	        IF #s_UDT_Status.Specific.ParcelTooLowError
	            OR #iqUDT_EquipmentControl.Command.ResetData
	        THEN
	            "FC_Statistics"(ix_Reset := #iqUDT_EquipmentControl.Command.ResetData,
	                            ix_Activate := #s_UDT_Status.Specific.ParcelTooLowError,
	                            ix_RTrigActivate := #s_R_TRIG_ParcelTooLow.Q,
	                            iqUDT_Statistics := #s_UDT_DimensionsCheckStatistics.TooLowParcels);
	        END_IF;

	    END_REGION

	    REGION 9.5 - Too wide parcels statistics

	        IF #s_UDT_Status.Specific.ParcelTooWideError
	            OR #iqUDT_EquipmentControl.Command.ResetData
	        THEN
	            "FC_Statistics"(ix_Reset := #iqUDT_EquipmentControl.Command.ResetData,
	                            ix_Activate := #s_UDT_Status.Specific.ParcelTooWideError,
	                            ix_RTrigActivate := #s_R_TRIG_ParcelTooWide.Q,
	                            iqUDT_Statistics := #s_UDT_DimensionsCheckStatistics.TooWideParcels);
	        END_IF;

	    END_REGION

	    REGION 9.6 - Too narrow parcels statistics

	        IF #s_UDT_Status.Specific.ParcelTooNarrowError
	            OR #iqUDT_EquipmentControl.Command.ResetData
	        THEN
	            "FC_Statistics"(ix_Reset := #iqUDT_EquipmentControl.Command.ResetData,
	                            ix_Activate := #s_UDT_Status.Specific.ParcelTooNarrowError,
	                            ix_RTrigActivate := #s_R_TRIG_ParcelTooNarrow.Q,
	                            iqUDT_Statistics := #s_UDT_DimensionsCheckStatistics.TooNarrowParcels);
	        END_IF;

	    END_REGION

	    REGION 9.7 - Incorrect parcel orientation statistics

	        IF #s_UDT_Status.Specific.IncorrectParcelOrientationError
	            OR #iqUDT_EquipmentControl.Command.ResetData
	        THEN
	            "FC_Statistics"(ix_Reset := #iqUDT_EquipmentControl.Command.ResetData,
	                            ix_Activate := #s_UDT_Status.Specific.IncorrectParcelOrientationError,
	                            ix_RTrigActivate := #s_R_TRIG_IncorrectShape.Q,
	                            iqUDT_Statistics := #s_UDT_DimensionsCheckStatistics.IncorrectShape);
	        END_IF;

	    END_REGION

	    REGION 9.8 - General error statistics

	        IF #s_UDT_Status.Specific.GeneralError
	            OR #iqUDT_EquipmentControl.Command.ResetData
	        THEN
	            "FC_Statistics"(ix_Reset := #iqUDT_EquipmentControl.Command.ResetData,
	                            ix_Activate := #s_UDT_Status.Specific.GeneralError,
	                            ix_RTrigActivate := #s_R_TRIG_GeneralError.Q,
	                            iqUDT_Statistics := #s_UDT_DimensionsCheckStatistics.GeneralError);
	        END_IF;

	    END_REGION

	END_REGION

	REGION 10 - Status

	    //Status
	    IF #iqUDT_EquipmentControl.Report.EnergySave
	    THEN
	        #s_UDT_Status.Status := "DB_HMIStatusConfiguration".EnergySave;
	    END_IF;

	    IF #iqUDT_EquipmentControl.Report.Running
	    THEN
	        #s_UDT_Status.Status := "DB_HMIStatusConfiguration".Running;
	    END_IF;

	    IF #iqUDT_EquipmentControl.Report.Stopped
	    THEN
	        #s_UDT_Status.Status := "DB_HMIStatusConfiguration".Stopped;
	    END_IF;

	    IF #s_UDT_Status.Specific.ParcelTooLongError
	        OR #s_UDT_Status.Specific.ParcelTooShortError
	        OR #s_UDT_Status.Specific.ParcelTooHighError
	        OR #s_UDT_Status.Specific.ParcelTooLowError
	        OR #s_UDT_Status.Specific.ParcelTooWideError
	        OR #s_UDT_Status.Specific.ParcelTooNarrowError
	        OR #s_UDT_Status.Specific.IncorrectParcelOrientationError
	        OR #s_UDT_Status.Specific.GeneralError

	    THEN
	        #s_UDT_Status.Status := "DB_HMIStatusConfiguration".DimensionError;
	    END_IF;

	(*    IF #iq_UDT_EquipmentControl.Report.SafetyStop
	    THEN
	        #s_UDT_Status.Status := "DB_HMIStatusConfiguration".SafetyStop;
	    END_IF; *)

	END_REGION

	REGION 11 - Update outputs

	    #qUDT_HMIStatus := #s_UDT_Status;
	    #qx_RequestHoldConveyor := (#sx_RequestHold AND NOT #sx_RequestRunReverse) OR #s_UDT_Status.Specific.GeneralError;
	    #qx_RequestRunReverseConveyor := #sx_RequestRunReverse;

	    //Column buzzer
	    #qx_BuzzerColumn := (#sx_ParcelRejecte AND "mx_Clock_1Hz") AND NOT #ix_ReverseRunButton;
	    //Column blue light
	    #qx_LightColumn := (#sx_ParcelRejecte AND "mx_Clock_1Hz") AND NOT #ix_ReverseRunButton;

	    //Button blue light
	    //Steady - Reset and restart line
	    //Blink - Restart not possible, sensor dimensioning check is still covered
	    #qx_LightResetButton := (#sx_ParcelRejecte AND "mx_Clock_1Hz") OR (NOT #sx_ParcelRejecte AND #sx_RequestHold);

	    //Data to HMI
	    //Sensor 1
	    #qUDT_HMIData.ActualSensor1 := #ii_DistanceSensor1;
	    #qUDT_HMIData.OffsetSensor1 := #si_Offset_DistanceSensor1;
	    #qUDT_HMIData.PositionSensor1 := #ii_DistanceSensor1 - #si_Offset_DistanceSensor1;

	    //Sensor 2
	    #qUDT_HMIData.ActualSensor2 := #ii_DistanceSensor2;
	    #qUDT_HMIData.OffsetSensor2 := #si_Offset_DistanceSensor2;
	    #qUDT_HMIData.PositionSensor2 := #ii_DistanceSensor2 - #si_Offset_DistanceSensor2;

	    #qUDT_HMIData.BeltWidth := INT_TO_UINT(#iUDT_DimensionsCheckConfiguration.Position.BeltWidth);


	    IF #s_F_TRIG_WaitForAllScanData.Q THEN
	        IF (#ss_Parcel.Size[0].Width < INT_TO_UINT(#iUDT_DimensionsCheckConfiguration.Position.BeltWidth)) THEN
	            #sui_ProductWidth := #ss_Parcel.Size[0].Width;
	        ELSE
	            #sui_ProductWidth := 0;
	        END_IF;

	        FOR #ti_LoopParcelLength := 0 TO #ci_MeasurementArraySize DO

	            IF (#ss_Parcel.Size[#ti_LoopParcelLength].Width > #sui_ProductWidth) AND (#ss_Parcel.Size[#ti_LoopParcelLength].Width < INT_TO_UINT(#iUDT_DimensionsCheckConfiguration.Position.BeltWidth)) THEN
	                #sui_ProductWidth := #ss_Parcel.Size[#ti_LoopParcelLength].Width;
	            END_IF;

	        END_FOR;

	    END_IF;

	    IF (#sui_ProductWidth > 0)
	        AND (#sui_ProductWidth < #iUDT_DimensionsCheckConfiguration.Position.BeltWidth)
	    THEN

	        #qUDT_HMIData.ProductWidth := #sui_ProductWidth;

	    ELSE

	        #qUDT_HMIData.ProductWidth := 0;

	    END_IF;

	END_REGION

	REGION 12 - Deactivation of functionality

	    #s_UDT_Status.Specific.DisabledGeneralFunctionality := #iUDT_DimensionsCheckCommand.DisableGeneral;
	    #s_UDT_Status.Specific.DisabledTooLongParcel := #iUDT_DimensionsCheckConfiguration.Functionality.TooLongParcelError AND #iUDT_DimensionsCheckCommand.DisableTooLongParcelError;
	    #s_UDT_Status.Specific.DisabledTooShortParcelError := #iUDT_DimensionsCheckConfiguration.Functionality.TooShortParcelError AND #iUDT_DimensionsCheckCommand.DisableTooShortParcelError;
	    #s_UDT_Status.Specific.DisabledTooHighParcelError := #iUDT_DimensionsCheckConfiguration.Functionality.TooHighParcelError AND #iUDT_DimensionsCheckCommand.DisableTooHighParcelError;
	    #s_UDT_Status.Specific.DisabledTooLowParcelError := #iUDT_DimensionsCheckConfiguration.Functionality.TooLowParcelError AND #iUDT_DimensionsCheckCommand.DisableTooLowParcelError;
	    #s_UDT_Status.Specific.DisabledTooWideParcelError := #iUDT_DimensionsCheckConfiguration.Functionality.TooWideParcelError AND #iUDT_DimensionsCheckCommand.DisableTooWideParcelError;
	    #s_UDT_Status.Specific.DisabledTooNarrowParcelError := #iUDT_DimensionsCheckConfiguration.Functionality.TooNarrowParcelError AND #iUDT_DimensionsCheckCommand.DisableTooNarrowParcelError;
	    #s_UDT_Status.Specific.DisabledParcelOrientationError := #iUDT_DimensionsCheckConfiguration.Functionality.ParcelOrientationError AND #iUDT_DimensionsCheckCommand.DisableParcelOrientationError;

	END_REGION
END_FUNCTION_BLOCK

FUNCTION_BLOCK "FB_PECUpdate"
TITLE = FB_PECUpdate
{ S7_Optimized_Access := 'TRUE' }
AUTHOR : MHSE
FAMILY : GeneralSystemFunctions
VERSION : 3.0
// ATTRIBUTES
// AUTO_NUMBER = True
// BLOCK_NUMBER = 221
// END_ATTRIBUTES
//Function block to update parcel data in a tracking array at PEC position.
   VAR_INPUT
      iUDT_PECUpdateConfiguration { ExternalAccessible := 'False'; ExternalVisible := 'False'; ExternalWritable := 'False'} : "UDT_PECUpdateConfiguration";   //   PEC update configuration
      iUDT_ConveyorCommonConfiguration { ExternalAccessible := 'False'; ExternalVisible := 'False'; ExternalWritable := 'False'} : "UDT_ConveyorCommonConfiguration";   //   Conveyor configuration
      ix_PEC { ExternalAccessible := 'False'; ExternalVisible := 'False'; ExternalWritable := 'False'} : Bool;   //   TRUE when the end of section photoeye is not blocked
      ix_TeachingMode { ExternalAccessible := 'False'; ExternalVisible := 'False'; ExternalWritable := 'False'} : Bool;   //   Teaching mode enable
   END_VAR

   VAR_OUTPUT
      qUDT_Status { ExternalAccessible := 'False'; ExternalVisible := 'False'; ExternalWritable := 'False'} : "UDT_PECUpdateStatus";   //   Status structure
      qi_GINwrite { ExternalAccessible := 'False'; ExternalVisible := 'False'; ExternalWritable := 'False'} : Int;   //  Gin found or generated
      qx_PECFiltered { ExternalAccessible := 'False'; ExternalVisible := 'False'; ExternalWritable := 'False'} : Bool;   //   Filtered photoeye signal
   END_VAR

   VAR_IN_OUT
      iqUDT_ConveyorInterface : "UDT_ConveyorInterface";   //   Conveyor interface
      iqUDT_UnknownGINRange : "UDT_UnknownGIN";   //   Unknown GIN
      iqUDT_FifoHeader : "UDT_FifoHeader";   //   FIFO header
      iqUDT_Statistics : "UDT_PECUpdateStatistics";   //   Statistic structure
      iqa_TrackingData : Array[*] of Int;   //   Tracking data
      iqa_FifoData : Array[*] of Int;   //   FIFO data
   END_VAR

   VAR
      sFB_PEC { ExternalAccessible := 'False'; ExternalVisible := 'False'; ExternalWritable := 'False'; S7_SetPoint := 'False'} : "FB_PEC";   //   Photoeye function
      sFB_LengthMeasurement { ExternalAccessible := 'False'; ExternalVisible := 'False'; ExternalWritable := 'False'; S7_SetPoint := 'False'} : "FB_ParcelLength";   //   Length measurement
      sUDT_LostGINFIFOStatus { ExternalAccessible := 'False'; ExternalVisible := 'False'; ExternalWritable := 'False'; S7_SetPoint := 'False'} : "UDT_FifoStatus";   //   Lost GIN FIFO status
      ss_PECDataDeviation { ExternalAccessible := 'False'; ExternalVisible := 'False'; ExternalWritable := 'False'} : Struct   // PEC/Data deviation calculation structure
         Last { ExternalAccessible := 'False'; ExternalVisible := 'False'; ExternalWritable := 'False'} : Int;   //  Last deviation [cm]
         GIN { ExternalAccessible := 'False'; ExternalVisible := 'False'; ExternalWritable := 'False'} : Int;   //  Last GIN deviation
         Sum { ExternalAccessible := 'False'; ExternalVisible := 'False'; ExternalWritable := 'False'} : Int;   //  Deviation sum [cm]
         Nr { ExternalAccessible := 'False'; ExternalVisible := 'False'; ExternalWritable := 'False'} : Int;   //  Deviation number
      END_STRUCT;
      ss_ValidGINRange { ExternalAccessible := 'False'; ExternalVisible := 'False'; ExternalWritable := 'False'} : Struct   //   Valid GIN range
         Start { ExternalAccessible := 'False'; ExternalVisible := 'False'; ExternalWritable := 'False'} : Int;
         End { ExternalAccessible := 'False'; ExternalVisible := 'False'; ExternalWritable := 'False'} : Int;
         GIN { ExternalAccessible := 'False'; ExternalVisible := 'False'; ExternalWritable := 'False'} : Int;
      END_STRUCT;
      ss_AlignedParcelsCounters { ExternalAccessible := 'False'; ExternalVisible := 'False'; ExternalWritable := 'False'} : Struct   //   Aligned parcels counters
         Total { ExternalAccessible := 'False'; ExternalVisible := 'False'; ExternalWritable := 'False'} : Int;   //   Total aligned parcels
         DataNoPEC { ExternalAccessible := 'False'; ExternalVisible := 'False'; ExternalWritable := 'False'} : Int;   //   Parcels aligned in case data detected without photoeye signal
         PECNoData { ExternalAccessible := 'False'; ExternalVisible := 'False'; ExternalWritable := 'False'} : Int;   //   Parcels aligned in case parcel detected without data
      END_STRUCT;
      ss_LostParcelsCounters { ExternalAccessible := 'False'; ExternalVisible := 'False'; ExternalWritable := 'False'} : Struct   //   Lost parcels counters
         Total { ExternalAccessible := 'False'; ExternalVisible := 'False'; ExternalWritable := 'False'} : Int;   //   Total number of lost parcels
         DoubleData { ExternalAccessible := 'False'; ExternalVisible := 'False'; ExternalWritable := 'False'} : Int;   //   Parcels lost due to double data found in a search window
         ParcelNotFound { ExternalAccessible := 'False'; ExternalVisible := 'False'; ExternalWritable := 'False'} : Int;   //   Parcels lost due to no parcel detected after travelling search window distance
      END_STRUCT;
      ss_LostValidParcelsCounters { ExternalAccessible := 'False'; ExternalVisible := 'False'; ExternalWritable := 'False'} : Struct   //   Lost parcels counters
         Total { ExternalAccessible := 'False'; ExternalVisible := 'False'; ExternalWritable := 'False'} : Int;   //   Total number of lost parcels
         DoubleData { ExternalAccessible := 'False'; ExternalVisible := 'False'; ExternalWritable := 'False'} : Int;   //   Parcels lost due to double data found in a search window
         ParcelNotFound { ExternalAccessible := 'False'; ExternalVisible := 'False'; ExternalWritable := 'False'} : Int;   //   Parcels lost due to no parcel detected after travelling search window distance
      END_STRUCT;
      si_UnknownParcelsCounters { ExternalAccessible := 'False'; ExternalVisible := 'False'; ExternalWritable := 'False'} : Struct   //   Unknown parcels counters
         Total { ExternalAccessible := 'False'; ExternalVisible := 'False'; ExternalWritable := 'False'} : Int;   //   Total number of unknown parcels
         LostParcelFound { ExternalAccessible := 'False'; ExternalVisible := 'False'; ExternalWritable := 'False'} : Int;   //   Parcel found with a lost data, unknown GIN created
         DataNotFound { ExternalAccessible := 'False'; ExternalVisible := 'False'; ExternalWritable := 'False'} : Int;   //   Data not found during search window scan
      END_STRUCT;
      sR_TRIG_Parcel {InstructionName := 'R_TRIG'; LibVersion := '1.0'; ExternalAccessible := 'False'; ExternalVisible := 'False'; ExternalWritable := 'False'; S7_SetPoint := 'False'} : R_TRIG;   //   Parcel detected rising edge to count parcels
      sR_TRIG_ParcelFound {InstructionName := 'R_TRIG'; LibVersion := '1.0'; ExternalAccessible := 'False'; ExternalVisible := 'False'; ExternalWritable := 'False'; S7_SetPoint := 'False'} : R_TRIG;   //   Parcel detected rising edge to update the PEC position tracking record
      sR_TRIG_DataFound {InstructionName := 'R_TRIG'; LibVersion := '1.0'; ExternalAccessible := 'False'; ExternalVisible := 'False'; ExternalWritable := 'False'; S7_SetPoint := 'False'} : R_TRIG;   //   Any data found at a PEC position rising edge
      sR_TRIG_PositiveDataFound {InstructionName := 'R_TRIG'; LibVersion := '1.0'; ExternalAccessible := 'False'; ExternalVisible := 'False'; ExternalWritable := 'False'; S7_SetPoint := 'False'} : R_TRIG;   //   Positive data found at a PEC position rising edge
      sR_TRIG_TeachMode {InstructionName := 'R_TRIG'; LibVersion := '1.0'; ExternalAccessible := 'False'; ExternalVisible := 'False'; ExternalWritable := 'False'; S7_SetPoint := 'False'} : R_TRIG;   //   Teaching mode activation rising edge
      sR_TRIG_TooManyLost {InstructionName := 'R_TRIG'; LibVersion := '1.0'; ExternalAccessible := 'False'; ExternalVisible := 'False'; ExternalWritable := 'False'; S7_SetPoint := 'False'} : R_TRIG;   //   Too many lost parcels error statistics trigger
      slr_Performance { ExternalAccessible := 'False'; ExternalVisible := 'False'; ExternalWritable := 'False'} : LReal := 100.0;   //   Update performance [%]
      sdi_TotalNumberOfParcels { ExternalAccessible := 'False'; ExternalVisible := 'False'; ExternalWritable := 'False'} : DInt;   //   Total number of parcels detected
      sdi_TotalNumberOfData { ExternalAccessible := 'False'; ExternalVisible := 'False'; ExternalWritable := 'False'} : DInt;   //   Total number of data detected
      si_PECPosition { ExternalAccessible := 'False'; ExternalVisible := 'False'; ExternalWritable := 'False'} : Int;   //   Photoeye position [cm]
      si_SearchWindow { ExternalAccessible := 'False'; ExternalVisible := 'False'; ExternalWritable := 'False'} : Int;   //   Data search distance from photoeye position [cm]
      si_GINToWrite { ExternalAccessible := 'False'; ExternalVisible := 'False'; ExternalWritable := 'False'} : Int;   //   Found or generated GIN, which will be used to update photoeye position in the tracking array
      si_PositionToUpdate { ExternalAccessible := 'False'; ExternalVisible := 'False'; ExternalWritable := 'False'} : Int;   //   Position in a tracking array to be updated
      si_Direction { ExternalAccessible := 'False'; ExternalVisible := 'False'; ExternalWritable := 'False'} : Int;   //   Direction of the displacement to parametrize loops
      si_Displacement { ExternalAccessible := 'False'; ExternalVisible := 'False'; ExternalWritable := 'False'} : Int;   //   Displacement [cm]
      si_ParcelWaitDistance { ExternalAccessible := 'False'; ExternalVisible := 'False'; ExternalWritable := 'False'} : Int;   //   Parcel delay [cm]
      si_LastUpdatedGIN { ExternalAccessible := 'False'; ExternalVisible := 'False'; ExternalWritable := 'False'} : Int;   //   Last updated GIN to check if next data is a new one
      si_LastCountedData { ExternalAccessible := 'False'; ExternalVisible := 'False'; ExternalWritable := 'False'} : Int;   //   Last counted data
      si_LostParcelsInARow { ExternalAccessible := 'False'; ExternalVisible := 'False'; ExternalWritable := 'False'} : Int;   //   Number of lost parcel in a row
      si_NumberOfTeachedParcels { ExternalAccessible := 'False'; ExternalVisible := 'False'; ExternalWritable := 'False'} : Int;   //   Number of teached parcels
      si_AverageSlip { ExternalAccessible := 'False'; ExternalVisible := 'False'; ExternalWritable := 'False'} : Int;   //   Average parcel slip [cm]
      si_CalculatedLengthCorrection { ExternalAccessible := 'False'; ExternalVisible := 'False'; ExternalWritable := 'False'} : Int;   //   Calculated length correction after teaching
      si_ParcelLengthFilterCounter { ExternalAccessible := 'False'; ExternalVisible := 'False'; ExternalWritable := 'False'} : Int;   //  Parcel length filter counter [cm]
      si_ParcelLengthFilterOldGIN { ExternalAccessible := 'False'; ExternalVisible := 'False'; ExternalWritable := 'False'} : Int;   //  Parcel length filter old GIN
      si_LoopCounter { ExternalAccessible := 'False'; ExternalVisible := 'False'; ExternalWritable := 'False'} : Int;   //   Loop counter
      sx_ParcelDetected { ExternalAccessible := 'False'; ExternalVisible := 'False'; ExternalWritable := 'False'} : Bool;   //   Parcel detected
      sx_ParcelWaitEnable { ExternalAccessible := 'False'; ExternalVisible := 'False'; ExternalWritable := 'False'} : Bool;   //   Missing parcel monitoring
      sx_TeachingMode { ExternalAccessible := 'False'; ExternalVisible := 'False'; ExternalWritable := 'False'} : Bool;   //   Teaching mode
      sx_GenerateGIN { ExternalAccessible := 'False'; ExternalVisible := 'False'; ExternalWritable := 'False'} : Bool;   //   Request to generate GIN
      sx_LostGINFIFOError { ExternalAccessible := 'False'; ExternalVisible := 'False'; ExternalWritable := 'False'} : Bool;   //   Lost GIN FIFO error
      sx_LostGINFIFOWarning { ExternalAccessible := 'False'; ExternalVisible := 'False'; ExternalWritable := 'False'} : Bool;   //   Lost GIN FIFO warning
      sx_InvalidDirection { ExternalAccessible := 'False'; ExternalVisible := 'False'; ExternalWritable := 'False'} : Bool;   //   Invalid direction
      sx_InvalidGINRange { ExternalAccessible := 'False'; ExternalVisible := 'False'; ExternalWritable := 'False'} : Bool;   //   Invalid GIN range
      sx_InvalidDisplacement { ExternalAccessible := 'False'; ExternalVisible := 'False'; ExternalWritable := 'False'} : Bool;   //   Invalid displacement
      sx_InvalidSearchWindow { ExternalAccessible := 'False'; ExternalVisible := 'False'; ExternalWritable := 'False'} : Bool;   //   Invalid search window
      sx_DoubleDataFound { ExternalAccessible := 'False'; ExternalVisible := 'False'; ExternalWritable := 'False'} : Bool;   //   Double data detected
      sx_LengthMeasurementEnable { ExternalAccessible := 'False'; ExternalVisible := 'False'; ExternalWritable := 'False'} : Bool;
   END_VAR

   VAR_TEMP
      tUDT_PECConfiguration : "UDT_PECConfiguration";   //   PEC configuration
      tUDT_PECStatus : "UDT_PECStatus";   //   PEC status
   END_VAR

   VAR CONSTANT
      ci_ZeroGIN : Int;   //   GIN = 0
   END_VAR


BEGIN
	(*
	----------------------------------------------------------------------------------------

	Version history:
	Date        | Version   | Author        | Remark
	----------------------------------------------------------------------------------------
	24/05/2019  | 0.1       | L.Klar        | first release MHSE TIA 15.1
	13/06/2019  | 0.2       | A.Nowak       | Replacement of instruction if for direct write into variable
	21/06/2019  | 0.3       | A.Nowak       | Add gap mesurement function and reorganise block (regions)
	24/07/2019  | 2.0       | L.Klar        | 2.0 MHSE library release TIA 15.1
	23/08/2019  | 2.1       | L.Klar        | "UDT_ConveyorConfiguration" changed to "UDT_ConveyorCommonConfiguration"
	XX/08/2019  | 2.2       | L.Klar        | Update logic changed
	19/09/2019  | 2.3       | P.Majka       | Updating checking PEC and PEC filtered signals
	30/09/2019  | 2.4       | L.Klar        | FB_PEC added, Filtered PEC signal output added
	21/10/2019  | 2.6       | L.Klar        | Configuration UDT chanaged to input, PEC configuration interface input name changed
	23/10/2019  | 2.7       | P.Majka       | Added Region 1, renumerating Regions, changed logic in Region 10.3 and Region 5
	29/10/2019  | 2.8       | L.Klar        | FB_PEC call changed
	14/11/2019  | 2.9       | L.Klar        | Deviations calculation corrected
	14/11/2019  | 3.0       | P.Majka       | 3.0 MHSE library release TIA 15.1
	20/12/2019  | 3.1       | S.Deulkar     | Used configureation error bit to report to conveyor block
	07/01/2020  | 3.2       | L.Klar        | GIN record structure updated, GIN cleared with default one during generation
	                                        | PECUpdate configuration UDT update - search window DINT -> INT,
	                                        | Conveyor common configuration UDT update - length INT -> DINT  conversion added
	29/01/2020  | 3.3       | L.Klar        | Negative GIN handling fixed, configuration bit added to delete negative GIN instead of ignoing it.
	24/02/2020  | 3.4       | L.Klar        | Formating changes, statistics counter added
	10/03/2020  | 3.5       | F.Baten       | Range check unknown GIN region 7
	26/03/2020  | 3.6       | F.Baten       | Added output 'qi_GINwrite'
	25/11/2020  | 3.7       | L.Klar        | Length filter added
	07/12/2020  | 3.8       | L.Klar        | Length filter bug fix
	22/01/2021  | 3.9       | L.Klar        | Total number of parcels and lost parcels counter fixed
	14/08/2021  | 3.10      | S. Deulkar    | Update from EMA
	21/02/2023  | 4.0       | F.Baten       | 4.0 Release TIA 17.5
	*)


	REGION 1 – FIFO header status update

	    "FC_Fifo"(ic_Mode := 'S',
	              qUDT_Status => #sUDT_LostGINFIFOStatus,
	              qx_Error => #sx_LostGINFIFOError,
	              qx_Warning => #sx_LostGINFIFOWarning,
	              iqv_Data := #si_GINToWrite,
	              iqUDT_FifoHeader := #iqUDT_FifoHeader,
	              iqv_DataBuffer := #iqa_FifoData);

	END_REGION

	REGION 2 – Displacement read

	    #si_Displacement := #iqUDT_ConveyorInterface.Displacement;

	END_REGION

	REGION 3 – PEC Position conversion from mm to cm

	    // The conversion is required because the photoeye position is given in mm and the tracking resolution is 1 cm.
	    #si_PECPosition := DINT_TO_INT(#iUDT_PECUpdateConfiguration.Distance / 10);

	END_REGION

	REGION 4 – Teaching mode enable

	    (* Teaching mode is used to calculate conveyor length correction, which allows to align real conveyor length with a tracking array length.
	       Correction is calculated as a difference between photoeye signal and tracking data deviations.
	       Calculated correction has to be manually copied from a FB_PECUpdate instance data block to conveyor configuration.*)

	    // Teaching mode is initialized and activated manually via block input.
	    #sR_TRIG_TeachMode(CLK := #ix_TeachingMode);

	    IF (#sR_TRIG_TeachMode.Q
	        AND NOT #sx_TeachingMode)
	    THEN
	        #ss_PECDataDeviation.Nr := 0;
	        #ss_PECDataDeviation.Sum := 0;
	        #si_NumberOfTeachedParcels := 0;
	        #sx_TeachingMode := TRUE;
	    END_IF;

	END_REGION

	REGION 5 – Photoeye

	    (*FB_PEC block call to filter photoeye signal and calculate jam status.*)

	    // Copy PEC configuration.
	    #tUDT_PECConfiguration.Distance := #iUDT_PECUpdateConfiguration.Distance;
	    #tUDT_PECConfiguration.JamDisplacementLimit := #iUDT_PECUpdateConfiguration.JamDisplacementLimit;
	    #tUDT_PECConfiguration.TimeOnDelay := #iUDT_PECUpdateConfiguration.TimeOnDelay;
	    #tUDT_PECConfiguration.TimeOffDelay := #iUDT_PECUpdateConfiguration.TimeOffDelay;
	    #tUDT_PECConfiguration.ResetWithPECBlocked := #iUDT_PECUpdateConfiguration.ResetWithPECBlocked;

	    //Call FB_PEC.
	    #sFB_PEC(ix_PEC := #ix_PEC,
	             iUDT_PECConfiguration := #tUDT_PECConfiguration,
	             qUDT_HMIStatus => #tUDT_PECStatus,
	             iqUDT_ConveyorInterface := #iqUDT_ConveyorInterface,
	             iqUDT_PECStatistics := #iqUDT_Statistics.PEC);

	    // Parcel length filter
	    IF NOT #ix_PEC
	        AND #iUDT_PECUpdateConfiguration.ParcelLengthFilter
	        AND #iqa_TrackingData[#si_PECPosition - 1] > 0
	        AND #iqa_TrackingData[#si_PECPosition - 1] <> #si_ParcelLengthFilterOldGIN THEN

	        IF "DB_GIN".GIN[#iqa_TrackingData[#si_PECPosition - 1]].General.Length > 0 THEN
	            #si_ParcelLengthFilterCounter := "DB_GIN".GIN[#iqa_TrackingData[#si_PECPosition - 1]].General.Length;
	        END_IF;

	        #si_ParcelLengthFilterOldGIN := #iqa_TrackingData[#si_PECPosition - 1];

	    END_IF;

	    IF #si_ParcelLengthFilterCounter > 0 THEN

	        #qUDT_Status.PEC := FALSE;
	        #qx_PECFiltered := FALSE;
	        #si_ParcelLengthFilterCounter -= #iqUDT_ConveyorInterface.Displacement;

	    ELSE

	        #qUDT_Status.PEC := #sFB_PEC.qx_PECFiltered;
	        #qx_PECFiltered := #sFB_PEC.qx_PECFiltered;

	    END_IF;

	    #qUDT_Status.Jam := #tUDT_PECStatus.Jam;

	    // Parcel detected variable to simplify further photoeye position tracking record update.
	    #sx_ParcelDetected := NOT #qUDT_Status.PEC;

	END_REGION

	REGION 6 – Error reset

	    // Reset errors when reset signal is given.
	    IF (#iqUDT_ConveyorInterface.InternalErrorReset)
	    THEN
	        #si_LostParcelsInARow := 0;
	        #qUDT_Status.TooManyLost := FALSE;
	        #sx_InvalidDisplacement := FALSE;
	    END_IF;

	END_REGION

	REGION 7 – GIN generator initialization

	    // Valid GIN range configuration is moved to a structure.
	    #ss_ValidGINRange.Start := #iUDT_PECUpdateConfiguration.GINRangeStart;
	    #ss_ValidGINRange.End := #iUDT_PECUpdateConfiguration.GINRangeEnd;

	    // Check if the unknown GIN is within range
	    IF #iqUDT_UnknownGINRange.GIN < #iqUDT_UnknownGINRange.Start
	        OR #iqUDT_UnknownGINRange.GIN > #iqUDT_UnknownGINRange.End
	    THEN
	        #iqUDT_UnknownGINRange.GIN := #iqUDT_UnknownGINRange.Start;
	    END_IF;

	    // Whenever valid GIN range is changed and the generated GIN doesn't fit, it's initialized.
	    IF (#ss_ValidGINRange.GIN < #ss_ValidGINRange.Start
	        OR #ss_ValidGINRange.GIN > #ss_ValidGINRange.End)
	    THEN
	        #ss_ValidGINRange.GIN := #ss_ValidGINRange.Start;
	    END_IF;

	    // Valid GIN range is set locally in PEC update configuration structure and it can't overlap with a global unknown GIN range.
	    #sx_InvalidGINRange := #iUDT_PECUpdateConfiguration.GenerationPoint
	    AND (#ss_ValidGINRange.End <= #ss_ValidGINRange.Start
	    OR #ss_ValidGINRange.Start <= #iqUDT_UnknownGINRange.End
	    OR #iqUDT_UnknownGINRange.End <= #iqUDT_UnknownGINRange.Start)
	    AND #ss_ValidGINRange.Start < 1000;   // Until 1000 it is UFO range

	END_REGION

	REGION 8 – Search window and displacement validation

	    (*Both parameters have to be checked to prevent tracking array exceeding.*)

	    // Search window cannot be lower than zero and greater than distance between PEC position and conveyor edge.
	    #sx_InvalidSearchWindow := #iUDT_PECUpdateConfiguration.SearchWindowFwd < 0
	    OR #iUDT_PECUpdateConfiguration.SearchWindowFwd >= #iUDT_ConveyorCommonConfiguration.Length + #iUDT_ConveyorCommonConfiguration.LengthCorrection - #si_PECPosition
	    OR #iUDT_PECUpdateConfiguration.SearchWindowRvs < 0
	    OR #iUDT_PECUpdateConfiguration.SearchWindowRvs >= #si_PECPosition;

	    // Displacement cannot be greater than the photoeye position.
	    IF (ABS(#si_Displacement) > #si_PECPosition)
	    THEN
	        #sx_InvalidDisplacement := TRUE;
	    END_IF;

	END_REGION

	REGION 9 – Total number of parcels counter

	    (*Parcels are counted basing on parcel detection rising edge trigger. Counting is blocked
	      during PLC first scan, when photoeye signal becomes 0.*)

	    #sR_TRIG_Parcel(CLK := #sx_ParcelDetected);

	    IF (#sR_TRIG_Parcel.Q
	        AND NOT "DB_Memory".FirstScan)
	    THEN
	        // Total number of parcels.
	        #sdi_TotalNumberOfParcels += 1;

	        // Every detected parcel resets lost parcels in a row counter.
	        #si_LostParcelsInARow := 0;

	        // Number of teached parcels is incremented if teaching mode is activated.
	        IF (#sx_TeachingMode)
	        THEN
	            #si_NumberOfTeachedParcels += 1;
	        END_IF;
	    END_IF;

	END_REGION

	REGION 10 – PEC Update
	    (* Photoeye position record is updated after every tracking register shift, basing on
	       actual situation - photoeye signal and data availability. In case of displacement
	       graeter than one, the loop will be executed the proper number of times. The update loop
	       can be executed if there is no configuration errors and the displacement was given.*)

	    WHILE #si_Displacement <> 0
	        AND NOT #sx_InvalidGINRange
	        AND NOT #sx_InvalidDisplacement
	        AND NOT #sx_InvalidSearchWindow
	    DO

	        REGION 10.1 – Direction

	            (*Depending on displacement sign, the direction of movement is determinated. This allows to choose
	            ` correct search window and parametrize all search loops to count up or down.*)

	            IF (#si_Displacement < 0)
	            THEN
	                #si_Direction := -1;
	                #si_SearchWindow := #iUDT_PECUpdateConfiguration.SearchWindowRvs;
	            ELSIF (#si_Displacement > 0)
	            THEN
	                #si_Direction := 1;
	                #si_SearchWindow := #iUDT_PECUpdateConfiguration.SearchWindowFwd;
	            END_IF;

	        END_REGION

	        REGION 10.2 – Position to update

	            // Position pointer used to specify the tracking array record to be updated.
	            #si_PositionToUpdate := #si_PECPosition - #si_Displacement + #si_Direction;

	        END_REGION


	        REGION 10.3 – Total number of data counter

	            (*Total number of data is incremented every time when new GIN is detected.*)

	            IF (#iqa_TrackingData[#si_PositionToUpdate + 1] > 0
	                AND #iqa_TrackingData[#si_PositionToUpdate + 1] <> #si_LastCountedData)
	            THEN
	                #sdi_TotalNumberOfData += 1;
	                #si_LastCountedData := #iqa_TrackingData[#si_PositionToUpdate + 1];
	            END_IF;

	        END_REGION

	        REGION 10.4 – GIN detection

	            (* Data found and parcel found triggers are used to determine the update case,
	               whether the data occurred first or a parcel.*)

	            // Trigger on any data found at a PEC position to detect the front of the parcel data.
	            #sR_TRIG_DataFound(CLK := #iqa_TrackingData[#si_PositionToUpdate] <> 0);

	            // Trigger on positive data found at a PEC position to detect the front of the parcel data.
	            #sR_TRIG_PositiveDataFound(CLK := #iqa_TrackingData[#si_PositionToUpdate] > 0);

	            // Trigger to detect front of the parcel.
	            #sR_TRIG_ParcelFound(CLK := #sx_ParcelDetected);

	(*
	Data detected without PEC signal

	                         Search window
	                          <--------|
	Data                              PEC
	|----------------------------------|------------------------------------------|
	|                           XXXXXXXX                                          |
	|----------------------------------|------------------------------------------|
	                                   |
	Conveyor                           |
	|----------------------------------|------------------------------------------|
	|                      YYYYYYYY    |                                          |
	|                      YYYYYYYY    |                                          |
	|                      YYYYYYYY    |                                          |
	|----------------------------------|------------------------------------------|
	*)
	(* Data detected without PEC signal.*)
	            IF (#sR_TRIG_PositiveDataFound.Q
	                AND NOT #sx_ParcelDetected)
	            THEN
	                #si_GINToWrite := 0;
	                // Double data detection loop.
	                FOR #si_LoopCounter := #si_PositionToUpdate TO
	                    #si_PECPosition + (#si_SearchWindow * #si_Direction) BY #si_Direction DO
	                    // Data found in a search window.
	                    IF (#iqa_TrackingData[#si_LoopCounter] > 0)
	                    THEN
	                        // First GIN found.
	                        IF (#si_GINToWrite = 0)
	                        THEN
	                            // Get the GIN if it's different than last updated GIN.
	                            IF #iqa_TrackingData[#si_LoopCounter] <> #si_LastUpdatedGIN THEN
	                                #si_GINToWrite := #iqa_TrackingData[#si_LoopCounter];
	                            END_IF;
	                            // If the first GIN was found, the scan loop conitues to check if there is no other data.
	                        ELSE
	                            // Next found data is different than the first one. Double data detected.
	                            IF (#iqa_TrackingData[#si_LoopCounter] <> #si_GINToWrite)
	                            THEN
	                                #sx_DoubleDataFound := TRUE;
	                                // First found GIN is marked as a lost one and the GIN is stored in a FIFO register.
	                                IF ("DB_GIN".GIN[#si_GINToWrite].General.Lost = FALSE)
	                                THEN
	                                    "DB_GIN".GIN[#si_GINToWrite].General.Lost := TRUE;

	                                    "FC_Fifo"(ic_Mode := 'W',
	                                              qUDT_Status => #sUDT_LostGINFIFOStatus,
	                                              qx_Error => #sx_LostGINFIFOError,
	                                              qx_Warning => #sx_LostGINFIFOWarning,
	                                              iqv_Data := #si_GINToWrite,
	                                              iqUDT_FifoHeader := #iqUDT_FifoHeader,
	                                              iqv_DataBuffer := #iqa_FifoData);

	                                    // Update statistics
	                                    #ss_LostParcelsCounters.Total += 1;
	                                    #ss_LostParcelsCounters.DoubleData += 1;


	                                    ////////////////////

	                                    IF #si_GINToWrite >= 1000 THEN
	                                        #ss_LostValidParcelsCounters.Total += 1;
	                                        #ss_LostValidParcelsCounters.DoubleData += 1;
	                                    END_IF;

	                                    ////////////////
	                                END_IF;

	                                // Second found GIN is marked as a lost one and the GIN is stored in a FIFO register.
	                                IF ("DB_GIN".GIN[#iqa_TrackingData[#si_LoopCounter]].General.Lost = FALSE)
	                                THEN
	                                    "DB_GIN".GIN[#iqa_TrackingData[#si_LoopCounter]].General.Lost := TRUE;

	                                    "FC_Fifo"(ic_Mode := 'W',
	                                              qUDT_Status => #sUDT_LostGINFIFOStatus,
	                                              qx_Error => #sx_LostGINFIFOError,
	                                              qx_Warning => #sx_LostGINFIFOWarning,
	                                              iqv_Data := #iqa_TrackingData[#si_LoopCounter],
	                                              iqUDT_FifoHeader := #iqUDT_FifoHeader,
	                                              iqv_DataBuffer := #iqa_FifoData);

	                                    // Update statistics
	                                    #ss_LostParcelsCounters.Total += 1;
	                                    #ss_LostParcelsCounters.DoubleData += 1;

	                                    ////////////////////

	                                    IF #iqa_TrackingData[#si_LoopCounter] >= 1000 THEN
	                                        #ss_LostValidParcelsCounters.Total += 1;
	                                        #ss_LostValidParcelsCounters.DoubleData += 1;
	                                    END_IF;

	                                    ////////////////
	                                    //
	                                END_IF;
	                                // Stop search window scan in case of double data detection
	                                EXIT;
	                            END_IF;
	                        END_IF;
	                    END_IF;
	                END_FOR;

	                // Becasue the data was found as a first one, GIN is stored and the logic to wait for a parcel is enebaled.
	                // If the double data was found there is no need to wait for a parcel. Data has been marked as a lost one.
	                IF NOT #sx_DoubleDataFound
	                THEN
	                    #sx_ParcelWaitEnable := TRUE;
	                END_IF;

	                #sx_DoubleDataFound := FALSE;
	(*
	Data and PEC signal detected at the same time - perfect match

	                         Search window
	                          <--------|
	Data                              PEC
	|----------------------------------|------------------------------------------|
	|                           XXXXXXXX                                          |
	|----------------------------------|------------------------------------------|
	                                   |
	Conveyor                           |
	|----------------------------------|------------------------------------------|
	|                           XXXXXXXX                                          |
	|                           XXXXXXXX                                          |
	|                           XXXXXXXX                                          |
	|----------------------------------|------------------------------------------|

	or PEC signal found without data or with old ones

	                         Search window
	                          <--------|
	Data                              PEC
	|----------------------------------|------------------------------------------|
	|                    XXXXXXXX      |                                          |
	|----------------------------------|------------------------------------------|
	                                   |
	Conveyor                           |
	|----------------------------------|------------------------------------------|
	|                           XXXXXXXX                                          |
	|                           XXXXXXXX                                          |
	|                           XXXXXXXX                                          |
	|----------------------------------|------------------------------------------|
	*)
	(*Data and PEC signal detected at the same time (perfect match) or PEC signal found without data or with old ones.*)
	            ELSIF (#sR_TRIG_ParcelFound.Q
	                AND (#sR_TRIG_PositiveDataFound.Q
	                OR (#iqa_TrackingData[#si_PositionToUpdate] = 0
	                OR #iqa_TrackingData[#si_PositionToUpdate] = #si_LastUpdatedGIN)
	                AND NOT #sx_ParcelWaitEnable))
	            THEN
	                // If the PEC is set as a GIN generation point, skip data detection loop and go to GIN generator.
	                IF (#iUDT_PECUpdateConfiguration.GenerationPoint)
	                THEN
	                    #sx_GenerateGIN := TRUE;
	                    // If the the PEC isn't a generation point, data search loop is enabled.
	                ELSE
	                    #si_GINToWrite := 0;

	                    // Double data detection loop.
	                    FOR #si_LoopCounter := #si_PositionToUpdate TO
	                        #si_PECPosition + (#si_SearchWindow * #si_Direction) BY #si_Direction DO

	                        // Data found in a search window.
	                        IF (#iqa_TrackingData[#si_LoopCounter] > 0)
	                        THEN
	                            // First GIN found.
	                            IF (#si_GINToWrite = 0)
	                            THEN
	                                // Get the GIN if it's different than last updated GIN.
	                                IF #iqa_TrackingData[#si_LoopCounter] <> #si_LastUpdatedGIN THEN
	                                    #si_GINToWrite := #iqa_TrackingData[#si_LoopCounter];

	                                    // PEC/Data deviation acquisition
	                                    #ss_PECDataDeviation.Last := DINT_TO_INT(#si_PECPosition - #si_LoopCounter);
	                                    #ss_PECDataDeviation.GIN := #si_GINToWrite;
	                                    #ss_PECDataDeviation.Sum -= ABS(#ss_PECDataDeviation.Last);
	                                    #ss_PECDataDeviation.Nr += 1;

	                                    // Parcel aligned statistics
	                                    IF (ABS(#ss_PECDataDeviation.Last) > ABS(#si_Displacement - 1))
	                                    THEN
	                                        #ss_AlignedParcelsCounters.Total += 1;
	                                        #ss_AlignedParcelsCounters.PECNoData += 1;
	                                    END_IF;
	                                END_IF;
	                                // If the first GIN was found, the scan loop conitues to check if there is no other data.
	                            ELSE
	                                // Next found data is different than the first one. Double data detected.
	                                IF (#iqa_TrackingData[#si_LoopCounter] <> #si_GINToWrite)
	                                THEN
	                                    // First found GIN is marked as a lost one and the GIN is stored in a FIFO register.
	                                    IF ("DB_GIN".GIN[#si_GINToWrite].General.Lost = FALSE)
	                                    THEN
	                                        "DB_GIN".GIN[#si_GINToWrite].General.Lost := TRUE;
	                                        "FC_Fifo"(ic_Mode := 'W',
	                                                  qUDT_Status => #sUDT_LostGINFIFOStatus,
	                                                  qx_Error => #sx_LostGINFIFOError,
	                                                  qx_Warning => #sx_LostGINFIFOWarning,
	                                                  iqv_Data := #si_GINToWrite,
	                                                  iqUDT_FifoHeader := #iqUDT_FifoHeader,
	                                                  iqv_DataBuffer := #iqa_FifoData);

	                                        // Update statistics
	                                        #ss_LostParcelsCounters.Total += 1;
	                                        #ss_LostParcelsCounters.DoubleData += 1;

	                                        ////////////////////

	                                        IF #si_GINToWrite >= 1000 THEN
	                                            #ss_LostValidParcelsCounters.Total += 1;
	                                            #ss_LostValidParcelsCounters.DoubleData += 1;
	                                        END_IF;

	                                        ////////////////
	                                        //
	                                    END_IF;

	                                    // Second found GIN is marked as a lost one and the GIN is stored in a FIFO register.
	                                    IF ("DB_GIN".GIN[#iqa_TrackingData[#si_LoopCounter]].General.Lost = FALSE)
	                                    THEN
	                                        "DB_GIN".GIN[#iqa_TrackingData[#si_LoopCounter]].General.Lost := TRUE;
	                                        "FC_Fifo"(ic_Mode := 'W',
	                                                  qUDT_Status => #sUDT_LostGINFIFOStatus,
	                                                  qx_Error => #sx_LostGINFIFOError,
	                                                  qx_Warning => #sx_LostGINFIFOWarning,
	                                                  iqv_Data := #iqa_TrackingData[#si_LoopCounter],
	                                                  iqUDT_FifoHeader := #iqUDT_FifoHeader,
	                                                  iqv_DataBuffer := #iqa_FifoData);

	                                        // Update statistics
	                                        #ss_LostParcelsCounters.Total += 1;
	                                        #ss_LostParcelsCounters.DoubleData += 1;

	                                        ////////////////////

	                                        IF #iqa_TrackingData[#si_LoopCounter] >= 1000 THEN
	                                            #ss_LostValidParcelsCounters.Total += 1;
	                                            #ss_LostValidParcelsCounters.DoubleData += 1;
	                                        END_IF;

	                                        ////////////////
	                                        //
	                                    END_IF;
	                                    // Stop search window scan in case of double data detection
	                                    EXIT;
	                                END_IF;
	                            END_IF;
	                        END_IF;
	                    END_FOR;

	                    // GIN not found in a search window
	                    IF (#si_GINToWrite = 0)
	                    THEN
	                        #sx_GenerateGIN := TRUE;
	                        #si_UnknownParcelsCounters.DataNotFound += 1;
	                    END_IF;

	                    // Found GIN is a lost one - generate unknown GIN
	                    // Found GIN isn't lost or it's negative - don't do anything
	                    IF (#si_GINToWrite > 0)
	                    THEN
	                        IF ("DB_GIN".GIN[#si_GINToWrite].General.Lost)
	                        THEN
	                            #sx_GenerateGIN := TRUE;
	                            #si_UnknownParcelsCounters.LostParcelFound += 1;
	                        END_IF;
	                    END_IF;
	                END_IF;

	                (*Second parcel has been found during data update. Situation can occur when search window is too short
	                  and the data is shifted. In that case found GIN will be marked as a lost one and new unknown GIN will be
	                  generated. Negative GIN will be ignored.*)
	            ELSIF (#sR_TRIG_ParcelFound.Q
	                AND (#iqa_TrackingData[#si_PositionToUpdate] <> 0
	                AND #iqa_TrackingData[#si_PositionToUpdate] <> #si_LastUpdatedGIN)
	                AND NOT #sx_ParcelWaitEnable)
	            THEN
	                IF (#iqa_TrackingData[#si_PositionToUpdate] > 0)
	                THEN
	                    IF ("DB_GIN".GIN[#iqa_TrackingData[#si_PositionToUpdate]].General.Lost = FALSE)
	                    THEN
	                        "DB_GIN".GIN[#iqa_TrackingData[#si_PositionToUpdate]].General.Lost := TRUE;
	                        "FC_Fifo"(ic_Mode := 'W',
	                                  qUDT_Status => #sUDT_LostGINFIFOStatus,
	                                  qx_Error => #sx_LostGINFIFOError,
	                                  qx_Warning => #sx_LostGINFIFOWarning,
	                                  iqv_Data := #iqa_TrackingData[#si_PositionToUpdate],
	                                  iqUDT_FifoHeader := #iqUDT_FifoHeader,
	                                  iqv_DataBuffer := #iqa_FifoData);

	                        // Update statistics
	                        #ss_LostParcelsCounters.Total += 1;
	                        #ss_LostParcelsCounters.DoubleData += 1;

	                        ////////////////////

	                        IF #iqa_TrackingData[#si_PositionToUpdate] >= 1000 THEN
	                            #ss_LostValidParcelsCounters.Total += 1;
	                            #ss_LostValidParcelsCounters.DoubleData += 1;
	                        END_IF;

	                        ////////////////
	                        //
	                    END_IF;
	                END_IF;

	                // Generate GIN
	                #sx_GenerateGIN := TRUE;
	                #si_UnknownParcelsCounters.LostParcelFound += 1;

	                (*Second data has been found during data update. Situation can occur when search window is too short
	                  and the data is shifted. In that case found GIN will be marked as a lost one.*)
	            ELSIF (#sR_TRIG_PositiveDataFound.Q
	                AND #sx_ParcelDetected
	                AND #iqa_TrackingData[#si_PositionToUpdate] <> #si_GINToWrite)
	            THEN
	                // Mark GIN as a lost one
	                IF ("DB_GIN".GIN[#iqa_TrackingData[#si_PositionToUpdate]].General.Lost = FALSE)
	                THEN
	                    "DB_GIN".GIN[#iqa_TrackingData[#si_PositionToUpdate]].General.Lost := TRUE;
	                    "FC_Fifo"(ic_Mode := 'W',
	                              qUDT_Status => #sUDT_LostGINFIFOStatus,
	                              qx_Error => #sx_LostGINFIFOError,
	                              qx_Warning => #sx_LostGINFIFOWarning,
	                              iqv_Data := #iqa_TrackingData[#si_PositionToUpdate],
	                              iqUDT_FifoHeader := #iqUDT_FifoHeader,
	                              iqv_DataBuffer := #iqa_FifoData);

	                    // Update statistics
	                    #ss_LostParcelsCounters.Total += 1;
	                    #ss_LostParcelsCounters.DoubleData += 1;

	                    ////////////////////

	                    IF #iqa_TrackingData[#si_PositionToUpdate] >= 1000 THEN
	                        #ss_LostValidParcelsCounters.Total += 1;
	                        #ss_LostValidParcelsCounters.DoubleData += 1;
	                    END_IF;

	                    ////////////////
	                END_IF;
	            END_IF;

	        END_REGION

	        REGION 10.5 – GIN generator

	            (*Used to generate new GIN. If the PEC position is a generation point, the number is taken from an internal GIN range.
	              If it's not, then GIN is taken from a global unknown GIN range.*)

	            IF (#sx_GenerateGIN)
	            THEN
	                // Generation point.
	                IF (#iUDT_PECUpdateConfiguration.GenerationPoint)
	                THEN
	                    // Generate GIN from a valid GIN range.
	                    IF (#ss_ValidGINRange.GIN <= #ss_ValidGINRange.End)
	                    THEN
	                        #si_GINToWrite := #ss_ValidGINRange.GIN;
	                        #ss_ValidGINRange.GIN += 1;
	                    ELSE
	                        #si_GINToWrite := #ss_ValidGINRange.Start;
	                        #ss_ValidGINRange.GIN := #ss_ValidGINRange.Start + 1;
	                    END_IF;
	                    // Unknown GIN generator.
	                ELSE
	                    // Generate GIN from a unknown GIN range.
	                    IF (#iqUDT_UnknownGINRange.GIN <= #iqUDT_UnknownGINRange.End)
	                    THEN
	                        #si_GINToWrite := #iqUDT_UnknownGINRange.GIN;
	                        #iqUDT_UnknownGINRange.GIN += 1;
	                    ELSE
	                        #si_GINToWrite := #iqUDT_UnknownGINRange.Start;
	                        #iqUDT_UnknownGINRange.GIN := #iqUDT_UnknownGINRange.Start + 1;
	                    END_IF;

	                    // Unknwn parcels statistics.
	                    #si_UnknownParcelsCounters.Total += 1;
	                END_IF;

	                // Reset generte GIN command.
	                #sx_GenerateGIN := FALSE;

	                // GIN record is cleared with configured default GIN record while it's generated.
	                "DB_GIN".GIN[#si_GINToWrite] := "DB_GINDefault".GIN[#iUDT_PECUpdateConfiguration.DefaultGIN];
	            END_IF;

	            #qi_GINwrite := #si_GINToWrite;

	        END_REGION


	        REGION 10.6 – PEC position data update

	            (*While parcel is detected, calculated GIN is written into the PEC position record.
	              If not, then the record is cleared with 0. Negative GIN is ignored or deleted, depending on configuration.*)

	            IF (#sx_ParcelDetected)
	            THEN

	                "FC_WriteGIN"(ii_GIN := #si_GINToWrite,
	                              ii_PositionToWrite := #si_PositionToUpdate,
	                              ii_NumberOfPositions := 1,
	                              ix_Direction := TRUE,
	                              iqa_TrackingData := #iqa_TrackingData);

	            ELSE
	                IF (#iqa_TrackingData[#si_PositionToUpdate] > 0
	                    OR #iUDT_PECUpdateConfiguration.NegativeGINDelete)
	                THEN

	                    "FC_WriteGIN"(ii_GIN := #ci_ZeroGIN,
	                                  ii_PositionToWrite := #si_PositionToUpdate,
	                                  ii_NumberOfPositions := 1,
	                                  ix_Direction := TRUE,
	                                  iqa_TrackingData := #iqa_TrackingData);

	                END_IF;
	            END_IF;

	        END_REGION

	        REGION 10.7 – Parcel waiting logic

	            (*Parcel waiting logic is used to wait for the photoeye signal for a search window distance.*)
	            IF (#sx_ParcelWaitEnable)
	            THEN
	                // Counting parcel wait distance depending on conveyor running direction if not detected.
	                IF (NOT #sx_ParcelDetected)
	                THEN
	                    IF (#si_Direction = 1)
	                    THEN
	                        #si_ParcelWaitDistance += 1;
	                    ELSE
	                        #si_ParcelWaitDistance -= 1;
	                    END_IF;

	                    // Parcel detected - stop waiting, use found GIN to update.
	                ELSE
	                    // PEC/Data deviation acquisition
	                    #ss_PECDataDeviation.Last := #si_ParcelWaitDistance;
	                    #ss_PECDataDeviation.GIN := #si_GINToWrite;
	                    #ss_PECDataDeviation.Sum += ABS(#ss_PECDataDeviation.Last);
	                    #ss_PECDataDeviation.Nr += 1;


	                    // Parcel aligned statistics
	                    IF (#ss_PECDataDeviation.Last > ABS(#si_Displacement - 1))
	                    THEN
	                        #ss_AlignedParcelsCounters.Total += 1;
	                        #ss_AlignedParcelsCounters.DataNoPEC += 1;
	                    END_IF;

	                    // Parcel waiting logic reset.
	                    #sx_ParcelWaitEnable := FALSE;
	                    #si_ParcelWaitDistance := 0;
	                END_IF;
	            END_IF;

	            // Parcel not found in a search window - stop waiting, mark found GIN as a lost one.
	            IF (ABS(#si_ParcelWaitDistance) = #si_SearchWindow)
	                AND (#si_GINToWrite > 0)
	            THEN
	                // Parcel lost
	                IF "DB_GIN".GIN[#si_GINToWrite].General.Lost = FALSE THEN
	                    "DB_GIN".GIN[#si_GINToWrite].General.Lost := TRUE;
	                    "FC_Fifo"(ic_Mode := 'W',
	                              qUDT_Status => #sUDT_LostGINFIFOStatus,
	                              qx_Error => #sx_LostGINFIFOError,
	                              qx_Warning => #sx_LostGINFIFOWarning,
	                              iqv_Data := #si_GINToWrite,
	                              iqUDT_FifoHeader := #iqUDT_FifoHeader,
	                              iqv_DataBuffer := #iqa_FifoData);

	                    // Parcel waiting logic reset.
	                    #si_ParcelWaitDistance := 0;
	                    #sx_ParcelWaitEnable := FALSE;

	                    // Lost parcels ina  row counter.
	                    #si_LostParcelsInARow += 1;

	                    // Update statistics.
	                    #ss_LostParcelsCounters.Total += 1;
	                    #ss_LostParcelsCounters.ParcelNotFound += 1;

	                    ////////////////////

	                    IF #si_GINToWrite >= 1000 THEN
	                        #ss_LostValidParcelsCounters.Total += 1;
	                        #ss_LostValidParcelsCounters.ParcelNotFound += 1;
	                    END_IF;

	                    ////////////////
	                    //
	                END_IF;

	            END_IF;

	            // Reset monitoring in case of going backwards.
	            IF (#si_ParcelWaitDistance = 0
	                AND NOT #sx_ParcelDetected
	                AND #sx_InvalidDirection)
	            THEN
	                #sx_ParcelWaitEnable := FALSE;
	            END_IF;

	            #sx_InvalidDirection := ((#si_Direction = 1
	            AND #si_ParcelWaitDistance < 0)
	            OR (#si_Direction = -1
	            AND #si_ParcelWaitDistance > 0));

	        END_REGION

	        REGION 10.8 – Last updated GIN

	            (*Last updated GIN to avoid processing the same data.*)
	            IF (#sR_TRIG_DataFound.Q)
	            THEN
	                #si_LastUpdatedGIN := #iqa_TrackingData[#si_PositionToUpdate];
	            END_IF;

	        END_REGION

	        REGION 10.8 – Update displacement

	            #si_Displacement := #si_Displacement - #si_Direction;

	        END_REGION

	    END_WHILE;

	END_REGION

	REGION 11 – Length measurement



	    (*Length and gap measurements can be enabled via PEC update configuration*)
	    #sFB_LengthMeasurement(ii_PECPosition := #si_PECPosition,
	                           ii_Displacement := #iqUDT_ConveyorInterface.Displacement,
	                           ix_LengthMeasurementEnable := #iUDT_PECUpdateConfiguration.ParcelLengthMeasurement OR #sx_LengthMeasurementEnable,
	                           ix_GapMeasurementEnable := #iUDT_PECUpdateConfiguration.GapLengthMeasurement,
	                           iqa_TrackingData := #iqa_TrackingData);

	    IF #iqa_TrackingData[#si_PECPosition] > 0
	        AND #iqa_TrackingData[#si_PECPosition] >= #iqUDT_UnknownGINRange.Start
	        AND #iqa_TrackingData[#si_PECPosition] <= #iqUDT_UnknownGINRange.End
	    THEN

	        #sx_LengthMeasurementEnable := "DB_GIN".GIN[#iqa_TrackingData[#si_PECPosition]].General.Length = 0;
	    ELSE

	        #sx_LengthMeasurementEnable := FALSE;

	    END_IF;

	END_REGION

	REGION 12 – Teaching done

	    // Average slip calculation
	    #si_AverageSlip := #ss_PECDataDeviation.Sum / #ss_PECDataDeviation.Nr;
	    #si_CalculatedLengthCorrection := DINT_TO_INT(#iUDT_ConveyorCommonConfiguration.LengthCorrection) + #si_AverageSlip * 10;
	    IF (#sx_TeachingMode                                                                                                            // Teaching mode enabled
	        AND #si_NumberOfTeachedParcels = #iUDT_PECUpdateConfiguration.NrOfTeachParcels)                                                 // Number of teaching parcels equal to the preset one                                                                                                                                                              // Teaching mode enabled ("sx_TeachMode")
	    THEN

	        #si_CalculatedLengthCorrection := DINT_TO_INT(#iUDT_ConveyorCommonConfiguration.LengthCorrection) + #si_AverageSlip * 10;
	        #sx_TeachingMode := FALSE;
	        #si_NumberOfTeachedParcels := 0;

	    END_IF;

	END_REGION

	REGION 13 – Performance

	    (*Performnce is a percentage ratio between number of lost parcels and total number of data, used to monitor data update efficiency.*)

	    IF (#sdi_TotalNumberOfData >= #ss_LostParcelsCounters.Total
	        AND #sdi_TotalNumberOfData > 0)
	    THEN
	        #slr_Performance := 100.0 - INT_TO_LREAL(#ss_LostParcelsCounters.Total) / #sdi_TotalNumberOfData * 100.0;
	    END_IF;

	    // Warning is generated if performance drops below 80%.
	    #qUDT_Status.LowPerformance := #slr_Performance < 80;

	END_REGION

	REGION 14 – Reset statistics

	    // Statistics are reset if reset signal is given.
	    IF #iqUDT_ConveyorInterface.ResetStatistics
	    THEN
	        #sdi_TotalNumberOfParcels := 0;
	        #ss_AlignedParcelsCounters.Total := 0;
	        #ss_AlignedParcelsCounters.PECNoData := 0;
	        #ss_AlignedParcelsCounters.DataNoPEC := 0;
	        #ss_LostParcelsCounters.Total := 0;
	        #ss_LostParcelsCounters.DoubleData := 0;
	        #ss_LostParcelsCounters.ParcelNotFound := 0;
	        #ss_LostValidParcelsCounters.Total := 0;
	        #ss_LostValidParcelsCounters.DoubleData := 0;
	        #ss_LostValidParcelsCounters.ParcelNotFound := 0;
	        #sdi_TotalNumberOfData := 0;
	        #si_UnknownParcelsCounters.Total := 0;
	        #si_UnknownParcelsCounters.LostParcelFound := 0;
	        #si_UnknownParcelsCounters.DataNotFound := 0;
	        #ss_PECDataDeviation.Sum := 0;
	        #ss_PECDataDeviation.Nr := 0;
	        #slr_Performance := 100;

	    END_IF;

	END_REGION

	REGION 15 – Too many lost parcels error

	    (*Error is generated if too many parcels will is marked as a lost one in a row*)
	    IF (#si_LostParcelsInARow >= #iUDT_PECUpdateConfiguration.MaxLost)
	    THEN
	        #qUDT_Status.TooManyLost := TRUE;
	    END_IF;

	END_REGION

	REGION 16 – Statistics

	    // Too many lost
	    #sR_TRIG_TooManyLost(CLK := #qUDT_Status.TooManyLost);
	    IF #qUDT_Status.TooManyLost
	        OR #iqUDT_ConveyorInterface.ResetStatistics
	    THEN
	        "FC_Statistics"(ix_Reset := #iqUDT_ConveyorInterface.ResetStatistics,
	                        ix_Activate := #qUDT_Status.TooManyLost,
	                        ix_RTrigActivate := #sR_TRIG_TooManyLost.Q,
	                        iqUDT_Statistics := #iqUDT_Statistics.TooManyLost);
	    END_IF;

	    // Total number of parcels
	    #iqUDT_Statistics.TotalNrOfParcels := #sdi_TotalNumberOfParcels;

	END_REGION

	REGION 17 – Internal tracking warning and error

	    // Internal tracking warning
	    IF (#qUDT_Status.LowPerformance
	        OR #sx_LostGINFIFOWarning)
	    THEN
	        #iqUDT_ConveyorInterface.InternalWarningTracking := TRUE;
	    END_IF;

	    // Internal tracking error
	    IF #qUDT_Status.TooManyLost
	    THEN
	        #iqUDT_ConveyorInterface.InternalErrorTracking := TRUE;
	    END_IF;

	    // Configuration error
	    IF (#sx_InvalidDisplacement
	        OR #sx_InvalidGINRange
	        OR #sx_InvalidSearchWindow)
	    THEN
	        #iqUDT_ConveyorInterface.ConfigurationError := TRUE;
	    END_IF;

	END_REGION
END_FUNCTION_BLOCK

FUNCTION_BLOCK "FB_PECBulk"
TITLE = FB_PEC
{ S7_Optimized_Access := 'TRUE' }
AUTHOR : MHSE
FAMILY : Conveyor
VERSION : 3.0
// ATTRIBUTES
// AUTO_NUMBER = True
// BLOCK_NUMBER = 220
// END_ATTRIBUTES
   VAR_INPUT
      ix_PEC { ExternalAccessible := 'False'; ExternalVisible := 'False'; ExternalWritable := 'False'} : Bool;   //   Signal of the PEC
      ix_PECDownstream { ExternalAccessible := 'False'; ExternalVisible := 'False'; ExternalWritable := 'False'} : Bool;   //   Downstream PEC signal
      ix_DownstreamRunning { ExternalAccessible := 'False'; ExternalVisible := 'False'; ExternalWritable := 'False'} : Bool;   //  Downstream conveyor is running
      iUDT_PECConfiguration { ExternalAccessible := 'False'; ExternalVisible := 'False'; ExternalWritable := 'False'} : "UDT_PECConfiguration";   //   PEC configuration structure
   END_VAR

   VAR_OUTPUT
      qx_PECFiltered { ExternalAccessible := 'False'; ExternalVisible := 'False'; ExternalWritable := 'False'} : Bool;   //   PEC Filtered
      qUDT_HMIStatus { ExternalAccessible := 'False'; ExternalVisible := 'False'; ExternalWritable := 'False'} : "UDT_PECStatus";   //   Status structure
   END_VAR

   VAR_IN_OUT
      iqUDT_ConveyorInterface : "UDT_ConveyorInterface";   //   Interface structure
      iqUDT_PECStatistics : "UDT_PECStatistics";   //   Statistics structure
   END_VAR

   VAR
      s_Status { ExternalAccessible := 'False'; ExternalVisible := 'False'; ExternalWritable := 'False'; S7_SetPoint := 'False'} : "UDT_PECStatus";   //   Status structure
      s_StatusOld { ExternalAccessible := 'False'; ExternalVisible := 'False'; ExternalWritable := 'False'; S7_SetPoint := 'False'} : "UDT_PECStatus";   //   Auxiliary status structure
      PEC_TimerOnOffDelay { ExternalAccessible := 'False'; ExternalVisible := 'False'; ExternalWritable := 'False'; S7_SetPoint := 'False'} : "FB_TimerOnOffDelay";   //   Filtering end of section photo eye signal
      sR_TRIG_PECJam {InstructionName := 'R_TRIG'; LibVersion := '1.0'; ExternalAccessible := 'False'; ExternalVisible := 'False'; ExternalWritable := 'False'; S7_SetPoint := 'False'} : R_TRIG;   //   Rising edge trigger PEC jam
   END_VAR
   VAR RETAIN
      si_AuxJamDisplacement { ExternalAccessible := 'False'; ExternalVisible := 'False'; ExternalWritable := 'False'} : Int;   //   Auxiliary variable to calculate displacement when PEC is blocked
   END_VAR
   VAR
      sx_Enable { ExternalAccessible := 'False'; ExternalVisible := 'False'; ExternalWritable := 'False'} : Bool;   //   Enable
      sx_PECFiltered { ExternalAccessible := 'False'; ExternalVisible := 'False'; ExternalWritable := 'False'} : Bool;   //   Photo eye filtered
   END_VAR


BEGIN
	(*
	----------------------------------------------------------------------------------------

	Version history:
	Date        | Version   | Author        | Remark
	----------------------------------------------------------------------------------------
	16/03/2020  | 3.0       | K.Pokorski    | 3.0 MHS library release TIA 15.1
	20/03/2020  | 3.1       | S.Theocharis  | Changed check to upsteam and jam condition
	24/03/2020  | 3.2       | S.Theocharis  | Add input ix Changed ix_UpstreamRunning
	30/03/2020  | 3.3       | K.Pokorski    | Changed error reset condition
	02/04/2020  | 3.4       | S.Theocharis  | Changed check to downsteam
	11/07/2022  | 3.5       | G.Vlooswijk   | Removed #ix_PECDownstream as jam reset condition
	21/02/2023  | 4.0       | F.Baten       | 4.0 Release TIA 17.5
	12/03/2024  | 4.1       | S. Nieswiec   | Small variable name changes according to current standard
	*)

	REGION 1 - Triggers

	    // Rising edge PEC Jam.
	    #sR_TRIG_PECJam(CLK := #s_Status.Jam);

	END_REGION

	REGION 2 - Active function

	    // To activate the Jam monitoring, the jam displacement limit must be greater than zero.
	    #sx_Enable := #iUDT_PECConfiguration.JamDisplacementLimit > 0;

	END_REGION

	REGION 3 - Reset errors

	    // Reset Jam error and initialize Jam displacement counter, when reset signal occurs.
	    IF #iqUDT_ConveyorInterface.InternalErrorReset
	        AND (#iUDT_PECConfiguration.ResetWithPECBlocked
	        OR (NOT #iUDT_PECConfiguration.ResetWithPECBlocked
	        AND #sx_PECFiltered))
	        AND #s_Status.Jam
	    THEN
	        #si_AuxJamDisplacement := 0;
	        #s_Status.Jam := FALSE;
	    END_IF;

	END_REGION

	REGION 4 - Photo eye filters

	    // End of section photo eye signal filter timer.
	    #PEC_TimerOnOffDelay(iudi_OnDelayTime := #iUDT_PECConfiguration.TimeOnDelay,
	                         iudi_OffDelayTime := #iUDT_PECConfiguration.TimeOffDelay,
	                         ix_SignalToDelay := #ix_PEC,
	                         ix_Enable := TRUE,
	                         qx_DelayedSignal => #sx_PECFiltered);

	    // Write the current status of the photo eye.
	    #s_Status.PEC := #sx_PECFiltered;
	    #qx_PECFiltered := #sx_PECFiltered;

	END_REGION

	REGION 5 - Jam detection

	    // Increasing Jam displacement counter by conveyor displacement, when photo eyes on conveyor and downstream conveyor are blocked and jam functionality is enable.
	    IF #ix_PECDownstream AND (NOT #sx_PECFiltered) AND #sx_Enable AND #ix_DownstreamRunning

	    THEN
	        #si_AuxJamDisplacement += #iqUDT_ConveyorInterface.Displacement;
	    ELSE
	        #si_AuxJamDisplacement := 0;
	    END_IF;

	    // Set jam error when total jam displacement exceeded limit.
	    IF (#si_AuxJamDisplacement > #iUDT_PECConfiguration.JamDisplacementLimit)
	        OR (#si_AuxJamDisplacement < (#iUDT_PECConfiguration.JamDisplacementLimit * -1))
	    THEN
	        #s_Status.Jam := TRUE;
	    END_IF;

	END_REGION

	REGION 6 - Statistics

	    // Jam Photo eye blocked statistics.
	    IF #s_Status.Jam
	        OR #iqUDT_ConveyorInterface.ResetStatistics
	    THEN
	        "FC_Statistics"(ix_Reset := #iqUDT_ConveyorInterface.ResetStatistics,
	                        ix_Activate := #s_Status.Jam,
	                        ix_RTrigActivate := #sR_TRIG_PECJam.Q,
	                        iqUDT_Statistics := #iqUDT_PECStatistics.Jam);
	    END_IF;

	END_REGION

	REGION 7 - Internal PEC error

	    // Set Internal photo eye error .
	    IF #s_Status.Jam
	    THEN
	        #iqUDT_ConveyorInterface.InternalErrorPEC := TRUE;
	    END_IF;

	END_REGION

	REGION 8 - Status

	    // Status update on change.
	    IF #s_StatusOld <> #s_Status
	    THEN
	        #qUDT_HMIStatus := #s_Status;
	        #s_StatusOld := #s_Status;
	    END_IF;

	END_REGION
END_FUNCTION_BLOCK

FUNCTION_BLOCK "FB_EuchnerLock"
{ S7_Optimized_Access := 'TRUE' }
VERSION : 0.1
// ATTRIBUTES
// AUTO_NUMBER = True
// BLOCK_NUMBER = 210
// END_ATTRIBUTES
   VAR_INPUT
      ix_ButtonReset { ExternalAccessible := 'False'; ExternalVisible := 'False'; ExternalWritable := 'False'} : Bool;   // Reset button
      ix_ButtonRequest { ExternalAccessible := 'False'; ExternalVisible := 'False'; ExternalWritable := 'False'} : Bool;   // Request open button
      ix_DoorClosed { ExternalAccessible := 'False'; ExternalVisible := 'False'; ExternalWritable := 'False'} : Bool;   // Feedback from lock - door is closed
      ix_BoltTongueClosed { ExternalAccessible := 'False'; ExternalVisible := 'False'; ExternalWritable := 'False'} : Bool;   // Feedback from lock - bolt tongue closed
      ix_SafelyLoced { ExternalAccessible := 'False'; ExternalVisible := 'False'; ExternalWritable := 'False'} : Bool;   // Feedback from lock - Safely locked
      ix_LockFault { ExternalAccessible := 'False'; ExternalVisible := 'False'; ExternalWritable := 'False'} : Bool;   // Lock has an internal fault
      ix_SystemStopped { ExternalAccessible := 'False'; ExternalVisible := 'False'; ExternalWritable := 'False'} : Bool;   // Feedback from system - System is stopped
      ix_SafetyLockOK { ExternalAccessible := 'False'; ExternalVisible := 'False'; ExternalWritable := 'False'} : Bool;   // Safety lock status OK
      ix_SafetyLockAckReq { ExternalAccessible := 'False'; ExternalVisible := 'False'; ExternalWritable := 'False'} : Bool;   // Safety lock need acknowledgement
   END_VAR

   VAR_OUTPUT
      qx_StopSystem { ExternalAccessible := 'False'; ExternalVisible := 'False'; ExternalWritable := 'False'} : Bool;   // Signal to stop the system
      qx_ResetButtonLed { ExternalAccessible := 'False'; ExternalVisible := 'False'; ExternalWritable := 'False'} : Bool;   // Reset button lamp
      qx_RequestButtonLed { ExternalAccessible := 'False'; ExternalVisible := 'False'; ExternalWritable := 'False'} : Bool;   // Request button lamp
      qx_FaultReset { ExternalAccessible := 'False'; ExternalVisible := 'False'; ExternalWritable := 'False'} : Bool;   // Reset internal lock fault
      qx_ReleaseLock { ExternalAccessible := 'False'; ExternalVisible := 'False'; ExternalWritable := 'False'} : Bool;   // Signal to safety logic to release lock
      qUDT_Status : "UDT_EuchnerLockStatus";   // Status structure
   END_VAR

   VAR
      sFB_OpenRequestDelay { ExternalAccessible := 'False'; ExternalVisible := 'False'; ExternalWritable := 'False'; S7_SetPoint := 'False'} : "FB_TimerOnOffDelay";   // Function block to generate on signal delay - emergency request button
      sFB_ResetDelay { ExternalAccessible := 'False'; ExternalVisible := 'False'; ExternalWritable := 'False'; S7_SetPoint := 'False'} : "FB_TimerOnOffDelay";
      sR_TRIG_RequestButton {InstructionName := 'R_TRIG'; LibVersion := '1.0'; ExternalAccessible := 'False'; ExternalVisible := 'False'; ExternalWritable := 'False'; S7_SetPoint := 'False'} : R_TRIG;   // Rising edge trigger from reqest button
      sx_Request { ExternalAccessible := 'False'; ExternalVisible := 'False'; ExternalWritable := 'False'} : Bool;   // Request to open the door
      sx_EmergencyReqest { ExternalAccessible := 'False'; ExternalVisible := 'False'; ExternalWritable := 'False'} : Bool;   // Emergency request to open the door
   END_VAR

   VAR CONSTANT
      c_Time : UDInt := 10000;
   END_VAR


BEGIN
	(*
	----------------------------------------------------------------------------------------

	Version history:
	Date        | Version   | Author        | Remark
	----------------------------------------------------------------------------------------
	11/03/2022  | 0.1       | S.Nikodem     | first release MHS TIA 15.1
	21/02/2023  | 4.0       | F.Baten       | 4.0 Release TIA 17.5
	*)

	REGION 1 - Request open

	    //Button
	    //Rising edge trigger
	    #sR_TRIG_RequestButton(CLK := #ix_ButtonRequest);

	    // Flip-flop
	    IF #sR_TRIG_RequestButton.Q THEN

	        IF #sx_Request THEN

	            #sx_Request := FALSE;
	            #sx_EmergencyReqest := FALSE;

	        ELSE

	            #sx_Request := TRUE;

	        END_IF;

	    END_IF;

	    // Reset Flip-Flop
	    IF NOT #ix_BoltTongueClosed THEN

	        #sx_Request := FALSE;
	        #sx_EmergencyReqest := FALSE;

	    END_IF;

	    //Emergency open reqest
	    #sFB_OpenRequestDelay(iudi_OnDelayTime := #c_Time,
	                          iudi_OffDelayTime := 0,
	                          ix_SignalToDelay := #ix_ButtonRequest,
	                          ix_Enable := True);


	    IF #sFB_OpenRequestDelay.qx_DelayedSignal THEN

	        #sx_EmergencyReqest := True;

	    END_IF;

	    //Stop system
	    #qx_StopSystem := #sx_Request OR #sx_EmergencyReqest;

	    //If system is stopped and is safe then open lock
	    #qx_ReleaseLock := (#sx_Request AND #ix_SystemStopped) OR #sx_EmergencyReqest;

	END_REGION

	REGION 2 - Lamp controlling

	    // Reset button LED - Blue
	    // Lamp active - Safety is open
	    // Lamp flashing - Euchner lock has a fault or safety lock must be acknowledged and bolt is inside.

	    #qx_ResetButtonLed := (NOT #ix_SafetyLockOK AND NOT #ix_SafetyLockAckReq) OR ("mx_Clock_1Hz" AND (#ix_SafetyLockAckReq OR #ix_LockFault));

	    // Request button LED - White
	    // Lamp active - Request to open the lock is active Aand lock is opened and bolt is inside.
	    // Lamp flashing - Request to open is active, the area is not safe and the lock is closed.

	    #qx_RequestButtonLed := #sx_Request AND ((NOT #ix_SafelyLoced AND #ix_BoltTongueClosed) OR "mx_Clock_1Hz");

	END_REGION

	REGION 3 - Falut reset

	    #sFB_ResetDelay(iudi_OnDelayTime := 0,
	                    iudi_OffDelayTime := 3500,
	                    ix_SignalToDelay := (#ix_LockFault) AND (#ix_ButtonReset));


	    // Set reset signal
	    #qx_FaultReset := #sFB_ResetDelay.qx_DelayedSignal;

	END_REGION

	REGION 4 - Status

	    // Copy status
	    #qUDT_Status.LockFault := #ix_LockFault;
	    #qUDT_Status.DoorClosed := #ix_DoorClosed;
	    #qUDT_Status.DoorOpened := NOT #ix_DoorClosed;
	    #qUDT_Status.BoltTongueClosed := #ix_BoltTongueClosed;
	    #qUDT_Status.Safelylocked := #ix_SafelyLoced;
	    #qUDT_Status.SafetyLockAckReq := #ix_SafetyLockAckReq;

	END_REGION

END_FUNCTION_BLOCK

FUNCTION_BLOCK "FB_MergeCapacity"
{ S7_Optimized_Access := 'TRUE' }
VERSION : 0.1
// ATTRIBUTES
// AUTO_NUMBER = True
// BLOCK_NUMBER = 218
// END_ATTRIBUTES
   VAR_INPUT
      ix_PEC_Merge { ExternalAccessible := 'False'; ExternalVisible := 'False'; ExternalWritable := 'False'} : Bool;
      iUDT_FlowConfig { ExternalAccessible := 'False'; ExternalVisible := 'False'; ExternalWritable := 'False'} : "UDT_FlowConfiguration" := ([6(1.0)], (), (), (), (), ());
      ix_XBSInductAvailable { ExternalAccessible := 'False'; ExternalVisible := 'False'; ExternalWritable := 'False'} : Bool;
   END_VAR

   VAR_OUTPUT
      qr_FlowCountMerge { ExternalAccessible := 'False'; ExternalVisible := 'False'; ExternalWritable := 'False'} : Real;
   END_VAR

   VAR_IN_OUT
      iqUDT_EquipmentControl : "UDT_EquipmentControl";
   END_VAR

   VAR
      s_R_TRIG_ParcelDetect_Merge {InstructionName := 'R_TRIG'; LibVersion := '1.0'; ExternalAccessible := 'False'; ExternalVisible := 'False'; ExternalWritable := 'False'; S7_SetPoint := 'False'} : R_TRIG;   //  Rising edge of PEC signal
      ss_CountingRegMerge { ExternalAccessible := 'False'; ExternalVisible := 'False'; ExternalWritable := 'False'} : Array[1..50] of Real;   //  Counting registers parcels
      s_FB_Pulse_TimerEndMergePeriod { ExternalAccessible := 'False'; ExternalVisible := 'False'; ExternalWritable := 'False'; S7_SetPoint := 'False'} : "FB_Pulse";
      sr_FlowMerge { ExternalAccessible := 'False'; ExternalVisible := 'False'; ExternalWritable := 'False'} : Real;
   END_VAR

   VAR_TEMP
      tx_EndMergePeriod : Bool;
   END_VAR


BEGIN
	(*
	----------------------------------------------------------------------------------------
	|                                                                                      |
	|  Copyright  2022             MHS                                                     |
	|  All Rights Reserved         Larenweg 90                                             |
	|                              5234 KC 's-Hertogenbosch,                               |
	|                              Netherlands                                             |
	|                                                                                      |
	----------------------------------------------------------------------------------------

	Version history:
	Date        | Version   | Author       | Remark
	----------------------------------------------------------------------------------------
	20/04/2022  | 3.0       | M.Roijen     | first release MHS TIA 15.1
	13/03/2024  | 4.1       | S.Nieswiec   | first release MHS TIA 18

	*)

	REGION 1 - Obtain capacity of Merge

	    // Rising edge PEC signal
	    #s_R_TRIG_ParcelDetect_Merge(CLK := #ix_PEC_Merge);

	    // Increase first counting register when new parcel detect
	    //
	    IF (#s_R_TRIG_ParcelDetect_Merge.Q)
	    THEN
	        #ss_CountingRegMerge[1] += 1;
	    END_IF;


	    #s_FB_Pulse_TimerEndMergePeriod(iudi_PulseTime := #iUDT_FlowConfig.PeriodMergeCapacity * 1000,
	                                    qx_Pulse => #tx_EndMergePeriod);

	    //Save capacity at the end of the period to array

	    IF (#tx_EndMergePeriod)
	    THEN

	        #sr_FlowMerge := (#ss_CountingRegMerge[1] / UDINT_TO_REAL(#iUDT_FlowConfig.PeriodMergeCapacity) * 3600);

	        IF NOT #ix_XBSInductAvailable THEN
	            #sr_FlowMerge := 0;
	        END_IF;

	        // Shifted counting register by one element down
	        MOVE_BLK(IN := #ss_CountingRegMerge[1],
	                 COUNT := 49,
	                 OUT => #ss_CountingRegMerge[2]);

	        // Reset first register
	        #ss_CountingRegMerge[1] := 0;

	    END_IF;



	END_REGION


	REGION 2 - Flow count reset

	    IF #iqUDT_EquipmentControl.Command.ResetData

	    THEN
	        FILL_BLK(IN := 0,
	                 COUNT := 50,
	                 OUT => #ss_CountingRegMerge[1]);
	        #sr_FlowMerge := 0;
	    END_IF;



	END_REGION


	REGION 3 - Write outputs

	    #qr_FlowCountMerge := #sr_FlowMerge;

	END_REGION

END_FUNCTION_BLOCK

FUNCTION_BLOCK "FB_FlowSplitter"
TITLE = Flow Splitter
{ S7_Optimized_Access := 'TRUE' }
AUTHOR : CLeite
VERSION : 3.0
// ATTRIBUTES
// AUTO_NUMBER = True
// BLOCK_NUMBER = 211
// END_ATTRIBUTES
   VAR_INPUT
      iUDT_FlowSplitterConfiguration { ExternalAccessible := 'False'; ExternalVisible := 'False'; ExternalWritable := 'False'} : "UDT_FlowSplitterConfiguration";   //  Flow splitter configuration structure
      iui_ExternalSpeed { ExternalAccessible := 'False'; ExternalVisible := 'False'; ExternalWritable := 'False'} : Int;   //  External speed [mm/s]
      ix_AirPressureOk { ExternalAccessible := 'False'; ExternalVisible := 'False'; ExternalWritable := 'False'} : Bool;   //  Air pressure circuit healthy
      ix_SafetyOk { ExternalAccessible := 'False'; ExternalVisible := 'False'; ExternalWritable := 'False'} : Bool;   //  TRUE when safety is ok
      ix_24vOk { ExternalAccessible := 'False'; ExternalVisible := 'False'; ExternalWritable := 'False'} : Bool;   //  TRUE when 24VDC is healthy
      ix_400vOk { ExternalAccessible := 'False'; ExternalVisible := 'False'; ExternalWritable := 'False'} : Bool;   //  TRUE when 400VAC is healthy
      ix_Connected { ExternalAccessible := 'False'; ExternalVisible := 'False'; ExternalWritable := 'False'} : Bool;   //  TRUE when the Isolator is electrically closed
      ix_HardwareOk { ExternalAccessible := 'False'; ExternalVisible := 'False'; ExternalWritable := 'False'} : Bool;   //   TRUE when  hardware is Ok
      ix_DebrisSensor { ExternalAccessible := 'False'; ExternalVisible := 'False'; ExternalWritable := 'False'} : Bool;   //  Signal from debris sensor
      ix_PECEos { ExternalAccessible := 'False'; ExternalVisible := 'False'; ExternalWritable := 'False'} : Bool;   //  End of section photo eye
      ix_PECUpstream { ExternalAccessible := 'False'; ExternalVisible := 'False'; ExternalWritable := 'False'} : Bool;   //  Upstream end of section photo eye
      ix_PECDivertChute { ExternalAccessible := 'False'; ExternalVisible := 'False'; ExternalWritable := 'False'} : Bool;   //  PEC of the divert chute
      ix_FlowSplitterEncoderError { ExternalAccessible := 'False'; ExternalVisible := 'False'; ExternalWritable := 'False'} : Bool;   //  True if there is an error with the flow splitter encoder
      ix_ExternalRequestHold { ExternalAccessible := 'False'; ExternalVisible := 'False'; ExternalWritable := 'False'} : Bool;   //  External request hold
      ix_HMICommunicationError { ExternalAccessible := 'False'; ExternalVisible := 'False'; ExternalWritable := 'False'} : Bool;   //  HMI Communication Error
      ix_ResetEnergySave { ExternalAccessible := 'False'; ExternalVisible := 'False'; ExternalWritable := 'False'} : Bool;   //   Reset save energy mode timer
   END_VAR

   VAR_OUTPUT
      qUDT_HMIStatus { ExternalAccessible := 'False'; ExternalVisible := 'False'; ExternalWritable := 'False'} : "UDT_FlowSplitterStatus";   //  HMI status structure
      qUDT_Status { ExternalAccessible := 'False'; ExternalVisible := 'False'; ExternalWritable := 'False'} : "UDT_CommonStatus";   //  Common status structure
      qx_Zone1Divert { ExternalAccessible := 'False'; ExternalVisible := 'False'; ExternalWritable := 'False'} : Bool;   //  Activation of the divert in zone divert side
      qx_Zone2Divert { ExternalAccessible := 'False'; ExternalVisible := 'False'; ExternalWritable := 'False'} : Bool;   //  Activation of the divert in zone straight side
   END_VAR

   VAR_IN_OUT
      iqUDT_EquipmentControl : "UDT_EquipmentControl";   //  Equipment control structure
      iqUDT_FlowSplitterCommand : "UDT_FlowSplitterCommand";   //  Flow splitter command structure
      iqUDT_FlowSplitterInterface : "UDT_ConveyorInterface";   //  Interface structure
      iqUDT_HandShakeUp : "UDT_ConveyorHandshake";   //  Handshake upstream structure
      iqUDT_HandShakeStraight : "UDT_ConveyorHandshake";   //  Handshake downstream straight structure
      iqUDT_HandShakeDivert : "UDT_ConveyorHandshake";   //  Handshake downstream divert structure
      iqUDT_Statistics : "UDT_FlowSplitterStatistics";   //  Statistics structure
   END_VAR

   VAR
      sUDT_CommonStatus { ExternalAccessible := 'False'; ExternalVisible := 'False'; ExternalWritable := 'False'; S7_SetPoint := 'False'} : "UDT_CommonStatus";   //  Common status structure
      sUDT_CommonStatusOld { ExternalAccessible := 'False'; ExternalVisible := 'False'; ExternalWritable := 'False'; S7_SetPoint := 'False'} : "UDT_CommonStatus";   //  Auxiliary status structure
      sUDT_HMIStatus { ExternalAccessible := 'False'; ExternalVisible := 'False'; ExternalWritable := 'False'; S7_SetPoint := 'False'} : "UDT_FlowSplitterStatus";   //  HMI status structure
      sFB_DebrisTimer { ExternalAccessible := 'False'; ExternalVisible := 'False'; ExternalWritable := 'False'; S7_SetPoint := 'False'} : "FB_TimerOnOffDelay";   //  Filtering debris photo eye signal
      sFB_CascadeModeTimer { ExternalAccessible := 'False'; ExternalVisible := 'False'; ExternalWritable := 'False'; S7_SetPoint := 'False'} : "FB_TimerOnOffDelay";   //  Timer to cascade start
      PEC_TimerOnOffDelay { ExternalAccessible := 'False'; ExternalVisible := 'False'; ExternalWritable := 'False'; S7_SetPoint := 'False'} : "FB_TimerOnOffDelay";   //  Timer to filter EOS PEC signal
      PEC_ChuteTimerOnOffDelay { ExternalAccessible := 'False'; ExternalVisible := 'False'; ExternalWritable := 'False'; S7_SetPoint := 'False'} : "FB_TimerOnOffDelay";   //  Timer to filter chute PEC signal
      PEC_UpstreamTimerOnOffDelay { ExternalAccessible := 'False'; ExternalVisible := 'False'; ExternalWritable := 'False'; S7_SetPoint := 'False'} : "FB_TimerOnOffDelay";   //  Timer to filter upstream PEC signal
      sFB_DivertsActivationTimer { ExternalAccessible := 'False'; ExternalVisible := 'False'; ExternalWritable := 'False'; S7_SetPoint := 'False'} : "FB_TimerOnOffDelay";   //  Timer to delay divert activation
      sR_TRIG_ManualMode {InstructionName := 'R_TRIG'; LibVersion := '1.0'; ExternalAccessible := 'False'; ExternalVisible := 'False'; ExternalWritable := 'False'; S7_SetPoint := 'False'} : R_TRIG;   //  Rising edge trigger manual mode
      sF_TRIG_ManualMode {InstructionName := 'F_TRIG'; LibVersion := '1.0'; ExternalAccessible := 'False'; ExternalVisible := 'False'; ExternalWritable := 'False'; S7_SetPoint := 'False'} : F_TRIG;   //  Falling edge trigger manual mode
      sR_TRIG_PECJam {InstructionName := 'R_TRIG'; LibVersion := '1.0'; ExternalAccessible := 'False'; ExternalVisible := 'False'; ExternalWritable := 'False'; S7_SetPoint := 'False'} : R_TRIG;   //  Rising edge trigger PEC jam
      sR_TRIG_PECDivertChuteJam {InstructionName := 'R_TRIG'; LibVersion := '1.0'; ExternalAccessible := 'False'; ExternalVisible := 'False'; ExternalWritable := 'False'; S7_SetPoint := 'False'} : R_TRIG;   //  Rising edge trigger PEC divert chute jam
      sR_TRIG_RunManual {InstructionName := 'R_TRIG'; LibVersion := '1.0'; ExternalAccessible := 'False'; ExternalVisible := 'False'; ExternalWritable := 'False'; S7_SetPoint := 'False'} : R_TRIG;   //  Rising edge run conveyor in manual mode
      sF_TRIG_RunManual {InstructionName := 'F_TRIG'; LibVersion := '1.0'; ExternalAccessible := 'False'; ExternalVisible := 'False'; ExternalWritable := 'False'; S7_SetPoint := 'False'} : F_TRIG;   //  Falling edge run conveyor in manual mode
      sR_TRIG_Jog {InstructionName := 'R_TRIG'; LibVersion := '1.0'; ExternalAccessible := 'False'; ExternalVisible := 'False'; ExternalWritable := 'False'; S7_SetPoint := 'False'} : R_TRIG;   //  Rising edge trigger manual jog
      sF_TRIG_Jog {InstructionName := 'F_TRIG'; LibVersion := '1.0'; ExternalAccessible := 'False'; ExternalVisible := 'False'; ExternalWritable := 'False'; S7_SetPoint := 'False'} : F_TRIG;   //  Falling edge trigger manual mode jog
      sR_TRIG_FlowSplitterUpTime {InstructionName := 'R_TRIG'; LibVersion := '1.0'; ExternalAccessible := 'False'; ExternalVisible := 'False'; ExternalWritable := 'False'; S7_SetPoint := 'False'} : R_TRIG;   //  Rising edge trigger flow splitter up time
      sR_TRIG_FlowSplitterDownTime {InstructionName := 'R_TRIG'; LibVersion := '1.0'; ExternalAccessible := 'False'; ExternalVisible := 'False'; ExternalWritable := 'False'; S7_SetPoint := 'False'} : R_TRIG;   //  Rising edge trigger flow splitter down
      sR_TRIG_AirPressureError {InstructionName := 'R_TRIG'; LibVersion := '1.0'; ExternalAccessible := 'False'; ExternalVisible := 'False'; ExternalWritable := 'False'; S7_SetPoint := 'False'} : R_TRIG;   //  Rising edge trigger air pressure error
      sR_TRIG_DebrisDetected {InstructionName := 'R_TRIG'; LibVersion := '1.0'; ExternalAccessible := 'False'; ExternalVisible := 'False'; ExternalWritable := 'False'; S7_SetPoint := 'False'} : R_TRIG;   //  Rising edge debris detected
      sR_TRIG_EnconderError {InstructionName := 'R_TRIG'; LibVersion := '1.0'; ExternalAccessible := 'False'; ExternalVisible := 'False'; ExternalWritable := 'False'; S7_SetPoint := 'False'} : R_TRIG;   //  Rising edge enconder error
      sR_TRIG_Mode1 {InstructionName := 'R_TRIG'; LibVersion := '1.0'; ExternalAccessible := 'False'; ExternalVisible := 'False'; ExternalWritable := 'False'; S7_SetPoint := 'False'} : R_TRIG;   //  Rising edge Mode 1 active
      sR_TRIG_Mode2 {InstructionName := 'R_TRIG'; LibVersion := '1.0'; ExternalAccessible := 'False'; ExternalVisible := 'False'; ExternalWritable := 'False'; S7_SetPoint := 'False'} : R_TRIG;   //  Rising edge Mode 2 active
      sR_TRIG_Mode3 {InstructionName := 'R_TRIG'; LibVersion := '1.0'; ExternalAccessible := 'False'; ExternalVisible := 'False'; ExternalWritable := 'False'; S7_SetPoint := 'False'} : R_TRIG;   //  Rising edge Mode 3 active
      sR_TRIG_Mode4 {InstructionName := 'R_TRIG'; LibVersion := '1.0'; ExternalAccessible := 'False'; ExternalVisible := 'False'; ExternalWritable := 'False'; S7_SetPoint := 'False'} : R_TRIG;   //  Rising edge Mode 4 active
      sR_TRIG_Mode5 {InstructionName := 'R_TRIG'; LibVersion := '1.0'; ExternalAccessible := 'False'; ExternalVisible := 'False'; ExternalWritable := 'False'; S7_SetPoint := 'False'} : R_TRIG;   //  Rising edge Mode 5 active
      sR_TRIG_EnergySave {InstructionName := 'R_TRIG'; LibVersion := '1.0'; ExternalAccessible := 'False'; ExternalVisible := 'False'; ExternalWritable := 'False'; S7_SetPoint := 'False'} : R_TRIG;   //  Rising edge trigger save energy mode active
   END_VAR
   VAR RETAIN
      si_AuxJamDisplacement { ExternalAccessible := 'False'; ExternalVisible := 'False'; ExternalWritable := 'False'} : Int;   //  Auxiliary jam displacement
      si_AuxJamDivertChuteDisplacement { ExternalAccessible := 'False'; ExternalVisible := 'False'; ExternalWritable := 'False'} : Int;   //  Divert chute displcement
      si_Mode { ExternalAccessible := 'False'; ExternalVisible := 'False'; ExternalWritable := 'False'} : Int;   //  Mode
      si_SwitchDelay { ExternalAccessible := 'False'; ExternalVisible := 'False'; ExternalWritable := 'False'} : Int;   //  Switch delay time
      si_Mode4AuxTimer { ExternalAccessible := 'False'; ExternalVisible := 'False'; ExternalWritable := 'False'} : Int;   //  Auxiliary variable to count time
      si_Mode4DivertTime { ExternalAccessible := 'False'; ExternalVisible := 'False'; ExternalWritable := 'False'} : Int;   //  Auxiliary variable divert time
   END_VAR
   VAR
      si_AuxEnergySave { ExternalAccessible := 'False'; ExternalVisible := 'False'; ExternalWritable := 'False'} : Int;   //   Auxinalary energy save
      sx_DebrisSignalFiltered { ExternalAccessible := 'False'; ExternalVisible := 'False'; ExternalWritable := 'False'} : Bool;   //  Debris detected
      sx_Ready { ExternalAccessible := 'False'; ExternalVisible := 'False'; ExternalWritable := 'False'} : Bool;   //  Flow splitter ready to operate in Automatic mode
   END_VAR
   VAR RETAIN
      sx_ManualModeActive { ExternalAccessible := 'False'; ExternalVisible := 'False'; ExternalWritable := 'False'} : Bool;   //  Manual mode active
      sx_StartReceived { ExternalAccessible := 'False'; ExternalVisible := 'False'; ExternalWritable := 'False'} : Bool;   //  Save start trigger from the system
      sx_AutomaticActive { ExternalAccessible := 'False'; ExternalVisible := 'False'; ExternalWritable := 'False'} : Bool;   //  Automatic active
   END_VAR
   VAR
      sx_PEC_EoSFiltered { ExternalAccessible := 'False'; ExternalVisible := 'False'; ExternalWritable := 'False'} : Bool;   //  End of section photo eye filtered
      sx_PEC_ChuteFiltered { ExternalAccessible := 'False'; ExternalVisible := 'False'; ExternalWritable := 'False'} : Bool;   //  Divert chute eye filtered
      sx_PEC_UpstreamFiltered { ExternalAccessible := 'False'; ExternalVisible := 'False'; ExternalWritable := 'False'} : Bool;   //  Upstream PEC filtered signal
   END_VAR
   VAR RETAIN
      sx_PreStartManual { ExternalAccessible := 'False'; ExternalVisible := 'False'; ExternalWritable := 'False'} : Bool;   //  Pre conditions to run conveyor in manual mode
      sx_Switch1To3 { ExternalAccessible := 'False'; ExternalVisible := 'False'; ExternalWritable := 'False'} : Bool;   //  Auxiliary bit when switch from mode 1 to 3
      sx_Switch3To1 { ExternalAccessible := 'False'; ExternalVisible := 'False'; ExternalWritable := 'False'} : Bool;   //  Auxiliary bit when switch from mode 3 to 1
      sx_Zone1_Divert { ExternalAccessible := 'False'; ExternalVisible := 'False'; ExternalWritable := 'False'} : Bool;   //  Static variable to active divert zone 1
      sx_Zone2_Divert { ExternalAccessible := 'False'; ExternalVisible := 'False'; ExternalWritable := 'False'} : Bool;   //  Static variable to active divert zone 2
      sx_EnableDiverts { ExternalAccessible := 'False'; ExternalVisible := 'False'; ExternalWritable := 'False'} : Bool;   //  When is true the diverts activation is enable
   END_VAR
   VAR
      sx_EnergySaveActive { ExternalAccessible := 'False'; ExternalVisible := 'False'; ExternalWritable := 'False'} : Bool;   //   Active energy save mode
   END_VAR

   VAR_TEMP
      tx_AuxBaseTimeDivert1 : Bool;   //  Temp variable to activate diverts zone 1
      tx_AuxBaseTimeDivert2 : Bool;   //  Temp variable to activate diverts zone 2
   END_VAR


BEGIN
	(*
	----------------------------------------------------------------------------------------

	Version history:
	Date        | Version   | Author        | Remark
	----------------------------------------------------------------------------------------
	//2019      | 1.0       | C.Leite       | first release TIA 15.1
	24/07/2019  | 2.0       | L.Klar        | 2.0 MHS library release TIA 15.1
	28/08/2019  | 2.1       | S.Deulkar     | modified fault logic, mode logic, reset logic
	                                        | And deleted sub region
	03/10/2019  | 2.2       | S.Deulkar     | Added comments
	03/10/2019  | 2.3       | S.Deulkar     | Updated UDT interface
	10/10/2019  | 2.4       | S. Deulkar    | Modified coulor status logic
	10/10/2019  | 2.5       | S. Deulkar    | Reverse logic is removed
	04/11/2019  | 2.6       | L.Klar        | 1 second pulse and frost scan changed from memory bit to DB variable
	12/11/2019  | 3.0       | P.Majka       | 3.0 MHS library release TIA 15.1
	20/12/2019  | 3.1       | S. Deulkar    | Added configuration error in make ready status
	11/01/2021  | 3.2       | L.Klar        | Input safety ok added to stop conveyor condition
	12/01/2021  | 3.3       | K. Pokorski   | Reset HMI commands of manual mode when conveyor no ready. Manual mode active to interface.
	12/01/2021  | 3.4       | S. Nikodem    | Added energy save mode
	04/02/2021  | 3.5       | K. Pokorski   | Status update fix
	17/02/2021  | 3.6       | K. Pokorski   | Internal error PEC handling
	02/03/2021  | 3.7       | K. Pokorski   | Halted status only if automatic on
	15/03/2021  | 3.8       | K. Pokorski   | Energy save corrected
	16/03/2021  | 3.9       | K. Pokorski   | On fly change mode corrected
	19/03/2021  | 3.10      | K.Pokorski    | Energy save pec eos changed
	21/02/2023  | 4.0       | F.Baten       | 4.0 Release TIA 17.5
	*)

	REGION 1 - Initial

	    // First PLC cycle
	    IF "DB_Memory".FirstScan
	    THEN
	        #sx_AutomaticActive := FALSE;                            // Automatic active
	        #iqUDT_HandShakeUp.RTR := False;                        // Reset RTR signal
	        #iqUDT_HandShakeUp.CascadeStartUp := FALSE;             // Reset cascade start signal
	        #iqUDT_FlowSplitterInterface.RunFwd := FALSE;           // Order to run forward to VFD
	        #iqUDT_FlowSplitterInterface.RunRvs := FALSE;           // Order to run reverse to VFD

	    END_IF;

	    // Mode selection
	    #si_Mode := #iqUDT_FlowSplitterCommand.Mode;                                   // Select mode from HMI inputs

	    IF (#si_Mode < 1) OR (#si_Mode > 5) OR #ix_HMICommunicationError THEN           // If there is no mode delected from HMI or HMI communication error is active
	        #si_Mode := #iUDT_FlowSplitterConfiguration.DefaultMode;                   // Select default mode from configuration
	    END_IF;

	    // Triggers
	    #sR_TRIG_ManualMode(CLK := #iqUDT_FlowSplitterCommand.ManualMode                // Rising edge trigger manual mode
	                        OR #iqUDT_EquipmentControl.Command.ManualMode);

	    #sF_TRIG_ManualMode(CLK := #iqUDT_FlowSplitterCommand.ManualMode                // Falling edge trigger manual mode
	                        OR #iqUDT_EquipmentControl.Command.ManualMode);

	    #sR_TRIG_Jog(CLK := #iqUDT_FlowSplitterCommand.ManualJog);                      // Rising edge trigger manual mode jog

	    #sF_TRIG_Jog(CLK := #iqUDT_FlowSplitterCommand.ManualJog);                      // Falling edge trigger manual mode jog

	    #sR_TRIG_RunManual(CLK := #iqUDT_FlowSplitterCommand.ManualStartStop);          // Rising edge trigger to start in manual mode

	    #sF_TRIG_RunManual(CLK := #iqUDT_FlowSplitterCommand.ManualStartStop);          // Falling edge trigger run in manual mode

	    #sR_TRIG_FlowSplitterUpTime(CLK := #sx_AutomaticActive AND #sx_Ready);           // Rising edge conveyor up

	    #sR_TRIG_PECJam(CLK := #sUDT_HMIStatus.Specific.PEC_EoSJam);                           // Rising edge PE Jam

	    #sR_TRIG_PECDivertChuteJam(CLK := #sUDT_HMIStatus.Specific.PEC_DivertChuteJam);        // Rising edge PE Jam

